//Scorer 7 - Axis positioning relative parameters
scorer7_AxisConfiguration.posRelative.distance := hmiCommands.slitter1.scorerPosCorrectionArr[7].positionCorrection;
scorer7_AxisConfiguration.posRelative.direction := 0;
scorer7_AxisConfiguration.posRelative.velocity := machineConfig.toolSlowPositioningVelocity;
scorer7_AxisConfiguration.posRelative.acceleration := machineConfig.toolSlowPositioningAccel;
scorer7_AxisConfiguration.posRelative.deceleration := machineConfig.toolFastPositioningAccel;
scorer7_AxisConfiguration.posRelative.jerk := machineConfig.toolSlowPositioningJerk;

//Scorer 7 - Axis JOG parameters
scorer7_AxisConfiguration.jog.velocity := machineConfig.toolSlowPositioningVelocity;
scorer7_AxisConfiguration.jog.acceleration := machineConfig.toolSlowPositioningAccel;
scorer7_AxisConfiguration.jog.deceleration := machineConfig.toolFastPositioningAccel;
scorer7_AxisConfiguration.jog.jerk := machineConfig.toolSlowPositioningJerk;

//Scorer 8
//_________________________________________________________________________________________________________________________

scorer8_AxisConfiguration.homing.position := machineConfig.homePositionScorer[8];
scorer8_AxisConfiguration.homing.offsetPosition := machineConfig.homePositionScorer[8];
scorer8_AxisConfiguration.homing.homeExecutionTimeLimit := T#5M;

scorer8_AxisConfiguration.posAbsolute.position := currentOrder.generatedOrder.scorerPositionReferenceArr[8] + machineConfig.scorerPositionCorrectionArr[8];
scorer8_AxisConfiguration.posAbsolute.velocity := machineConfig.toolFastPositioningVelocity;
scorer8_AxisConfiguration.posAbsolute.acceleration := machineConfig.toolFastPositioningAccel;
scorer8_AxisConfiguration.posAbsolute.deceleration := machineConfig.toolFastPositioningDecel;
scorer8_AxisConfiguration.posAbsolute.jerk := machineConfig.toolFastPositioningJerk;

//Scorer 8 - Axis positioning relative parameters
scorer8_AxisConfiguration.posRelative.distance := hmiCommands.slitter1.scorerPosCorrectionArr[8].positionCorrection;
scorer8_AxisConfiguration.posRelative.direction := 0;
scorer8_AxisConfiguration.posRelative.velocity := machineConfig.toolSlowPositioningVelocity;
scorer8_AxisConfiguration.posRelative.acceleration := machineConfig.toolSlowPositioningAccel;
scorer8_AxisConfiguration.posRelative.deceleration := machineConfig.toolFastPositioningAccel;
scorer8_AxisConfiguration.posRelative.jerk := machineConfig.toolSlowPositioningJerk;

//Scorer 8 - Axis JOG parameters
scorer8_AxisConfiguration.jog.velocity := machineConfig.toolSlowPositioningVelocity;
scorer8_AxisConfiguration.jog.acceleration := machineConfig.toolSlowPositioningAccel;
scorer8_AxisConfiguration.jog.deceleration := machineConfig.toolFastPositioningAccel;
scorer8_AxisConfiguration.jog.jerk := machineConfig.toolSlowPositioningJerk;

//----------------------------------------------------------------------------------------------
// Knife Axis control function block calls
//----------------------------------------------------------------------------------------------



IF executePositioning AND NOT executePositioningOld AND homeFinished THEN
//IF executePositioning AND NOT executePositioningOld THEN

	instFbCurrentOrderPositionsGeneration(execute := TRUE,
		machineConfig := machineConfig,
		currentOrder := currentOrder);
			
	IF NOT currentOrder.generatedOrder.statusWord.orderNotOk THEN
		
		instTONExecutePositioningDelay.IN := TRUE;
		positioningStarted	:= TRUE;

	END_IF

END_IF

executePositioningOld := executePositioning;

instTONExecutePositioningDelay(PT:=T#1S);



//Knife 1 - Axis control function block call
//__________________________________________________________________________
instFB_AxisControlKnife1_Axis(
    enable := TRUE,
	fastStop := haltAxis,
    enableAxis := enableAxis,
    resetAxis := resetCmd,
	posAbsolute := instTONExecutePositioningDelay.Q,
	posRelative	:= hmiCommands.slitter1.knifePosCorrectionArr[1].execute,
	jogForward := hmiCommands.slitter1.knifeJogArr[1].jogFw AND NOT homeSensorKnife2 AND homeFinished,
	jogBackward	:= hmiCommands.slitter1.knifeJogArr[1].jogRev AND NOT homeSensorKnife1 AND homeFinished,
    homingSensor := homeSensorKnife1,
    axis := knife1_Axis,
    master := knife1_Axis,
    configuration := knife1_AxisConfiguration
);

//Knife 2 - Axis control function block call
//__________________________________________________________________________

instFB_AxisControlKnife2_Axis(
    enable := TRUE,
	fastStop := haltAxis,	
    enableAxis := enableAxis,
    resetAxis := resetCmd,
	posAbsolute := instTONExecutePositioningDelay.Q,
	posRelative	:= hmiCommands.slitter1.knifePosCorrectionArr[2].execute,
	jogForward := hmiCommands.slitter1.knifeJogArr[2].jogFw AND NOT homeSensorKnife3 AND homeFinished,
	jogBackward	:= hmiCommands.slitter1.knifeJogArr[2].jogRev AND NOT homeSensorKnife2 AND homeFinished,
    homingSensor := homeSensorKnife2,
    axis := knife2_Axis,
    master := knife2_Axis,
    configuration := knife2_AxisConfiguration
);

//Knife 3 - Axis control function block call
//__________________________________________________________________________

instFB_AxisControlKnife3_Axis(
    enable := TRUE,
	fastStop := haltAxis,		
    enableAxis := enableAxis,
    resetAxis := resetCmd,
	posAbsolute := instTONExecutePositioningDelay.Q,
	posRelative	:= hmiCommands.slitter1.knifePosCorrectionArr[3].execute,
	jogForward := hmiCommands.slitter1.knifeJogArr[3].jogFw AND NOT (knife3_Axis.NcToPlc.ActPos > machineConfig.knifeMaxPostionArr[3]) AND NOT limitSensorKnife3_4 AND homeFinished,
	jogBackward	:= hmiCommands.slitter1.knifeJogArr[3].jogRev AND NOT homeSensorKnife3 AND homeFinished,
    homingSensor := homeSensorKnife3,
    axis := knife3_Axis,
    master := knife3_Axis,
    configuration := knife3_AxisConfiguration
);

//Knife 4 - Axis control function block call
//__________________________________________________________________________

instFB_AxisControlKnife4_Axis(
    enable := TRUE,
	fastStop := haltAxis,		
    enableAxis := enableAxis,
    resetAxis := resetCmd,
	posAbsolute := instTONExecutePositioningDelay.Q,
	posRelative	:= hmiCommands.slitter1.knifePosCorrectionArr[4].execute,
	jogForward := hmiCommands.slitter1.knifeJogArr[4].jogFw AND NOT homeSensorKnife4 AND homeFinished,
	jogBackward	:= hmiCommands.slitter1.knifeJogArr[4].jogRev AND NOT (knife4_Axis.NcToPlc.ActPos < machineConfig.knifeMinPostionArr[4]) AND NOT limitSensorKnife3_4 AND homeFinished,
    homingSensor := homeSensorKnife4,
    axis := knife4_Axis,
    master := knife4_Axis,
    configuration := knife4_AxisConfiguration
);

//Knife 5 - Axis control function block call
//__________________________________________________________________________

instFB_AxisControlKnife5_Axis(
    enable := TRUE,
	fastStop := haltAxis,		
    enableAxis := enableAxis,
    resetAxis := resetCmd,
	posAbsolute := instTONExecutePositioningDelay.Q,
	posRelative	:= hmiCommands.slitter1.knifePosCorrectionArr[5].execute,
	jogForward := hmiCommands.slitter1.knifeJogArr[5].jogFw AND NOT homeSensorKnife5 AND homeFinished,
	jogBackward	:= hmiCommands.slitter1.knifeJogArr[5].jogRev AND NOT homeSensorKnife4 AND homeFinished,
    homingSensor := homeSensorKnife5,
    axis := knife5_Axis,
    master := knife5_Axis,
    configuration := knife5_AxisConfiguration
);

//----------------------------------------------------------------------------------------------
// Scorer Axis control function block calls
//----------------------------------------------------------------------------------------------

//Scorer 1
//__________________________________________________________________________

instFB_AxisControlScorer1_Axis(
    enable := TRUE,
	fastStop := haltAxis,		
    enableAxis := enableAxis,
    resetAxis := resetCmd,
	posAbsolute := instTONExecutePositioningDelay.Q,
	posRelative	:= hmiCommands.slitter1.scorerPosCorrectionArr[1].execute,
	jogForward := hmiCommands.slitter1.scorerJogArr[1].jogFw AND NOT homeSensorScorer3 AND homeFinished,
	jogBackward	:= hmiCommands.slitter1.scorerJogArr[1].jogRev AND NOT homeSensorScorer1 AND homeFinished,
    homingSensor := homeSensorScorer1,
    axis := scorer1_Axis,
    master := scorer1_Axis,
    configuration := scorer1_AxisConfiguration
);
//Scorer 2
//__________________________________________________________________________

instFB_AxisControlScorer2_Axis(
    enable := TRUE,
	fastStop := haltAxis,		
    enableAxis := enableAxis,
    resetAxis := resetCmd,
	posAbsolute := instTONExecutePositioningDelay.Q,
	posRelative	:= hmiCommands.slitter1.scorerPosCorrectionArr[2].execute,
	jogForward := hmiCommands.slitter1.scorerJogArr[2].jogFw AND NOT homeSensorScorer4 AND homeFinished,
	jogBackward	:= hmiCommands.slitter1.scorerJogArr[2].jogRev AND NOT homeSensorScorer2 AND homeFinished,
    homingSensor := homeSensorScorer2,
    axis := scorer2_Axis,
    master := scorer2_Axis,
    configuration := scorer2_AxisConfiguration
);

//Scorer 3
//__________________________________________________________________________

instFB_AxisControlScorer3_Axis(
    enable := TRUE,
	fastStop := haltAxis,	
	
    enableAxis := enableAxis,
    resetAxis := resetCmd,
	posAbsolute := instTONExecutePositioningDelay.Q,
	posRelative	:= hmiCommands.slitter1.scorerPosCorrectionArr[3].execute,
	jogForward := hmiCommands.slitter1.scorerJogArr[3].jogFw AND NOT (scorer3_Axis.NcToPlc.ActPos > machineConfig.scorerMaxPostionArr[3]) AND NOT limitSensorScorer3_5 AND homeFinished,
	jogBackward	:= hmiCommands.slitter1.scorerJogArr[3].jogRev AND NOT homeSensorScorer3 AND homeFinished,
    homingSensor := homeSensorScorer3,
    axis := scorer3_Axis,
    master := scorer3_Axis,
    configuration := scorer3_AxisConfiguration
);

//Scorer 4
//__________________________________________________________________________

instFB_AxisControlScorer4_Axis(
    enable := TRUE,
	fastStop := haltAxis,	
	
    enableAxis := enableAxis,
    resetAxis := resetCmd,
	posAbsolute := instTONExecutePositioningDelay.Q,
	posRelative	:= hmiCommands.slitter1.scorerPosCorrectionArr[4].execute,
	jogForward := hmiCommands.slitter1.scorerJogArr[4].jogFw AND NOT (scorer4_Axis.NcToPlc.ActPos > machineConfig.scorerMaxPostionArr[4]) AND NOT limitSensorScorer4_6 AND homeFinished,
	jogBackward	:= hmiCommands.slitter1.scorerJogArr[4].jogRev AND NOT homeSensorScorer4 AND homeFinished,
    homingSensor := homeSensorScorer4,
    axis := scorer4_Axis,
    master := scorer4_Axis,
    configuration := scorer4_AxisConfiguration
);

//Scorer 5
//__________________________________________________________________________

instFB_AxisControlScorer5_Axis(
    enable := TRUE,
	fastStop := haltAxis,	
	
    enableAxis := enableAxis,
    resetAxis := resetCmd,
	posAbsolute := instTONExecutePositioningDelay.Q,
	posRelative	:= hmiCommands.slitter1.scorerPosCorrectionArr[5].execute,
	jogForward := hmiCommands.slitter1.scorerJogArr[5].jogFw AND NOT homeSensorScorer5 AND homeFinished,
	jogBackward	:= hmiCommands.slitter1.scorerJogArr[5].jogRev AND NOT (scorer5_Axis.NcToPlc.ActPos < machineConfig.scorerMinPostionArr[5]) AND NOT limitSensorScorer3_5 AND homeFinished,
    homingSensor := homeSensorScorer5,
    axis := scorer5_Axis,
    master := scorer5_Axis,
    configuration := scorer5_AxisConfiguration
);

//Scorer 6
//__________________________________________________________________________

instFB_AxisControlScorer6_Axis(
    enable := TRUE,
	fastStop := haltAxis,	
	
    enableAxis := enableAxis,
    resetAxis := resetCmd,
	posAbsolute := instTONExecutePositioningDelay.Q,
	posRelative	:= hmiCommands.slitter1.scorerPosCorrectionArr[6].execute,
	jogForward := hmiCommands.slitter1.scorerJogArr[6].jogFw AND NOT homeSensorScorer6 AND homeFinished,
	jogBackward	:= hmiCommands.slitter1.scorerJogArr[6].jogRev AND NOT (scorer6_Axis.NcToPlc.ActPos < machineConfig.scorerMinPostionArr[6]) AND NOT limitSensorScorer4_6 AND homeFinished,
    homingSensor := homeSensorScorer6,
    axis := scorer6_Axis,
    master := scorer6_Axis,
    configuration := scorer6_AxisConfiguration
);

//Scorer 7
//__________________________________________________________________________

instFB_AxisControlScorer7_Axis(
    enable := TRUE,
	fastStop := haltAxis,	
	
    enableAxis := enableAxis,
    resetAxis := resetCmd,
	posAbsolute := instTONExecutePositioningDelay.Q,
	posRelative	:= hmiCommands.slitter1.scorerPosCorrectionArr[7].execute,
	jogForward := hmiCommands.slitter1.scorerJogArr[7].jogFw AND NOT homeSensorScorer7 AND homeFinished,
	jogBackward	:= hmiCommands.slitter1.scorerJogArr[7].jogRev AND NOT homeSensorScorer5 AND homeFinished,
    homingSensor := homeSensorScorer7,
    axis := scorer7_Axis,
    master := scorer7_Axis,
    configuration := scorer7_AxisConfiguration
);

//Scorer 8
//__________________________________________________________________________

instFB_AxisControlScorer8_Axis(
    enable := TRUE,
	fastStop := haltAxis,	
	
    enableAxis := enableAxis,
    resetAxis := resetCmd,
	posAbsolute := instTONExecutePositioningDelay.Q,
	posRelative	:= hmiCommands.slitter1.scorerPosCorrectionArr[8].execute,
	jogForward := hmiCommands.slitter1.scorerJogArr[8].jogFw AND NOT homeSensorScorer8 AND homeFinished,
	jogBackward	:= hmiCommands.slitter1.scorerJogArr[8].jogRev AND NOT homeSensorScorer6 AND homeFinished,
    homingSensor := homeSensorScorer8,
    axis := scorer8_Axis,
    master := scorer8_Axis,
    configuration := scorer8_AxisConfiguration
);

IF instTONExecutePositioningDelay.Q THEN
	
	instTONExecutePositioningDelay.IN := FALSE;
	positioningStarted	:= FALSE;


END_IF
END_METHOD

METHOD PRIVATE _exhaustMotor
VAR_INPUT
END_VAR
(*
	startExhaustMotorCmd				: BOOL;
	stopExhaustMotorCmd				: BOOL;

*)

IF startExhaustMotorCmd AND safetyOK THEN
	
	startExhaustMotor := TRUE;


END_IF

IF stopExhaustMotorCmd THEN
	
	startExhaustMotor := FALSE;

END_IF



startExhaustMotorLamp := startExhaustMotor;
END_METHOD

METHOD PRIVATE _haltTheAxis
VAR_INPUT
END_VAR
(*

	homeSensorKnife1					: BOOL; // Knife 1 - Home sensor
	homeSensorKnife2					: BOOL; // Knife 2 - Home sensor
	homeSensorKnife3					: BOOL; // Knife 3 - Home sensor
	homeSensorKnife4					: BOOL; // Knife 4 - Home sensor
	homeSensorKnife5					: BOOL; // Knife 5 - Home sensor
	
	homeSensorScorer1					: BOOL; // Scorer 1 - Home sensor
	homeSensorScorer2					: BOOL; // Scorer 1 - Home sensor
	homeSensorScorer3					: BOOL; // Scorer 1 - Home sensor
	homeSensorScorer4					: BOOL; // Scorer 1 - Home sensor
	homeSensorScorer5					: BOOL; // Scorer 1 - Home sensor
	homeSensorScorer6					: BOOL; // Scorer 1 - Home sensor
	homeSensorScorer7					: BOOL; // Scorer 1 - Home sensor
	homeSensorScorer8					: BOOL; // Scorer 1 - Home sensor
*)

(*

	limitSensorKnife3_4					: BOOL;
	limitSensorScorer4_6					: BOOL;
	limitSensorScorer3_5					: BOOL;
*)
//-------------------------------------------------------------------------------------------------
// Halt Axis Logic: Prevent motion if any tool is detected on home sensor during active positioning
//-------------------------------------------------------------------------------------------------

// Activate the halt trigger if positioning is in progress 
// and any knife or scorer is detected in the home sensor
IF positioningRunning AND (
     homeSensorKnife1 OR
     homeSensorKnife2 OR
     homeSensorKnife3 OR
     homeSensorKnife4 OR
     homeSensorKnife5 OR
     homeSensorScorer1 OR
     homeSensorScorer2 OR
     homeSensorScorer3 OR
     homeSensorScorer4 OR
     homeSensorScorer5 OR
     homeSensorScorer6 OR
     homeSensorScorer7 OR
     homeSensorScorer8 OR
	 limitSensorKnife3_4 OR
	 limitSensorScorer3_5 OR
 	 limitSensorScorer4_6 
	 
) THEN
    instTPHaltAxis.IN := TRUE;
ELSE
    instTPHaltAxis.IN := FALSE;
END_IF

// Timer pulse for halting signal - triggers TRUE for 1 second
instTPHaltAxis(PT := T#1S);

// Output signal to halt all axes
haltAxis := instTPHaltAxis.Q;
END_METHOD

METHOD _homeFinished
VAR_INPUT
END_VAR
homeFinished := knife1_Axis.Status.Homed AND knife2_Axis.Status.Homed AND knife3_Axis.Status.Homed AND knife4_Axis.Status.Homed AND knife5_Axis.Status.Homed AND scorer1_Axis.Status.Homed AND scorer2_Axis.Status.Homed AND scorer3_Axis.Status.Homed AND scorer4_Axis.Status.Homed AND scorer5_Axis.Status.Homed AND scorer6_Axis.Status.Homed AND scorer7_Axis.Status.Homed AND scorer8_Axis.Status.Homed;
END_METHOD

METHOD PRIVATE _knifeLubrification
VAR_INPUT
END_VAR


(*
	knifeRunningMetersForSharpening		: ARRAY [1..5] OF INT;	(*This array is used to reset the lifetime meters that the knife runs*)
	knifeRunningMetersForLubfrication		: ARRAY [1..5] OF INT;	(*This array is used to reset the lifetime meters that the knife runs*)
	

*)

knifeLubrificationPump := startCutting;


instKnifeLubrificationCLK_PRG(PT:= T#1S, Q=> );


inst_FB_KnifeLubrification[1](
	machineRunning:= startTractionMotorCmd AND startCutting,
	manualLubrification := knife1LubrificationCmd, 
	measuringWheelSensor:= measuringWheelPulseSensor, 
	knifeEnabled:= knife1Enabled, 
	lubrificationSetpoint := machineConfig.knifeLubrificationDistance, 
	lubrificationTime:= machineConfig.knifeLubrificationTime, 
	lubrificationSolenoid=> knife1Lubrification);
	
inst_FB_KnifeLubrification[2](
	machineRunning:= startTractionMotorCmd AND startCutting,
	manualLubrification := knife2LubrificationCmd,  
	measuringWheelSensor:= measuringWheelPulseSensor, 
	knifeEnabled:= knife2Enabled, 
	lubrificationSetpoint := machineConfig.knifeLubrificationDistance, 
	lubrificationTime:= machineConfig.knifeLubrificationTime, 
	lubrificationSolenoid=> knife2Lubrification);
	
inst_FB_KnifeLubrification[3](
	machineRunning:= startTractionMotorCmd AND startCutting, 
	manualLubrification := knife3LubrificationCmd, 
	measuringWheelSensor:= measuringWheelPulseSensor, 
	knifeEnabled:= knife3Enabled, 
	lubrificationSetpoint := machineConfig.knifeLubrificationDistance, 
	lubrificationTime:= machineConfig.knifeLubrificationTime, 
	lubrificationSolenoid=> knife3Lubrification);	
	
inst_FB_KnifeLubrification[4](
	machineRunning:= startTractionMotorCmd AND startCutting, 
	manualLubrification := knife4LubrificationCmd, 	
	measuringWheelSensor:= measuringWheelPulseSensor, 
	knifeEnabled:= knife4Enabled, 
	lubrificationSetpoint := machineConfig.knifeLubrificationDistance, 
	lubrificationTime:= machineConfig.knifeLubrificationTime, 
	lubrificationSolenoid=> knife4Lubrification);		
	
	
inst_FB_KnifeLubrification[5](
	machineRunning:= startTractionMotorCmd AND startCutting, 
	manualLubrification := knife5LubrificationCmd,  
	measuringWheelSensor:= measuringWheelPulseSensor, 
	knifeEnabled:= knife5Enabled,
	lubrificationSetpoint := machineConfig.knifeLubrificationDistance, 
	lubrificationTime:= machineConfig.knifeLubrificationTime, 
	lubrificationSolenoid=> knife5Lubrification);		
	
arrKnifeRunningMetersForLubfrication[1] := inst_FB_KnifeLubrification[1].knifeRunningMeters;	
arrKnifeRunningMetersForLubfrication[2] := inst_FB_KnifeLubrification[2].knifeRunningMeters;	
arrKnifeRunningMetersForLubfrication[3] := inst_FB_KnifeLubrification[3].knifeRunningMeters;	
arrKnifeRunningMetersForLubfrication[4] := inst_FB_KnifeLubrification[4].knifeRunningMeters;	
arrKnifeRunningMetersForLubfrication[5] := inst_FB_KnifeLubrification[5].knifeRunningMeters;
END_METHOD

METHOD PRIVATE _knifeSharpening
VAR_INPUT
END_VAR
(*
	knifeRunningMetersForSharpening		: ARRAY [1..5] OF INT;	(*This array is used to reset the lifetime meters that the knife runs*)
	knifeRunningMetersForLubfrication		: ARRAY [1..5] OF INT;	(*This array is used to reset the lifetime meters that the knife runs*)
	

*)
//=================================================================================================
// KNIFE SHARPENING FB CALLS (1..7)
//=================================================================================================

inst_FB_KnifeSharpening[1](
    machineRunning        := knifeMotorStart,
    manualSharpening      := knifeManualSharpeningCmdArr[1],
    measuringWheelSensor  := measuringWheelPulseSensor,
    knifeEnabled          := currentOrder.generatedOrder.knifeEnabledArr[1],
    sharpeningSetpoint    := machineConfig.knifeSharpeningDistance,
    sharpeningTime        := machineConfig.knifeSharpeningTimeMS,
    sharpeningSolenoid    => knife1Sharpening
);

inst_FB_KnifeSharpening[2](
    machineRunning        := knifeMotorStart,
    manualSharpening      := knifeManualSharpeningCmdArr[2],
    measuringWheelSensor  := measuringWheelPulseSensor,
    knifeEnabled          := currentOrder.generatedOrder.knifeEnabledArr[2],
    sharpeningSetpoint    := machineConfig.knifeSharpeningDistance,
    sharpeningTime        := machineConfig.knifeSharpeningTimeMS,
    sharpeningSolenoid    => knife2Sharpening
);

inst_FB_KnifeSharpening[3](
    machineRunning        := knifeMotorStart,
    manualSharpening      := knifeManualSharpeningCmdArr[3],
    measuringWheelSensor  := measuringWheelPulseSensor,
    knifeEnabled          := currentOrder.generatedOrder.knifeEnabledArr[3],
    sharpeningSetpoint    := machineConfig.knifeSharpeningDistance,
    sharpeningTime        := machineConfig.knifeSharpeningTimeMS,
    sharpeningSolenoid    => knife3Sharpening
);

inst_FB_KnifeSharpening[4](
    machineRunning        := knifeMotorStart,
    manualSharpening      := knifeManualSharpeningCmdArr[4],
    measuringWheelSensor  := measuringWheelPulseSensor,
    knifeEnabled          := currentOrder.generatedOrder.knifeEnabledArr[4],
    sharpeningSetpoint    := machineConfig.knifeSharpeningDistance,
    sharpeningTime        := machineConfig.knifeSharpeningTimeMS,
    sharpeningSolenoid    => knife4Sharpening
);

inst_FB_KnifeSharpening[5](
    machineRunning        := knifeMotorStart,
    manualSharpening      := knifeManualSharpeningCmdArr[5],
    measuringWheelSensor  := measuringWheelPulseSensor,
    knifeEnabled          := currentOrder.generatedOrder.knifeEnabledArr[5],
    sharpeningSetpoint    := machineConfig.knifeSharpeningDistance,
    sharpeningTime        := machineConfig.knifeSharpeningTimeMS,
    sharpeningSolenoid    => knife5Sharpening
);
END_METHOD

METHOD PRIVATE _knifeSharpening_old
VAR_INPUT
END_VAR
(*
	knifeRunningMetersForSharpening		: ARRAY [1..5] OF INT;	(*This array is used to reset the lifetime meters that the knife runs*)
	knifeRunningMetersForLubfrication		: ARRAY [1..5] OF INT;	(*This array is used to reset the lifetime meters that the knife runs*)
	
	paperPresenceSensor				: BOOL;
	measuringWheelPaperPresenceSensor		: BOOL;
	rotaryShearCutPulse					: BOOL;	
	measuringWheelPulseSensor		: BOOL;	

*)

IF NOT knifeSharpeningAutoMan THEN
	
	knife1Sharpening := knife1SharpeningCmd;
	knife2Sharpening := knife2SharpeningCmd;
	knife3Sharpening := knife3SharpeningCmd;
	knife4Sharpening := knife4SharpeningCmd;
	knife5Sharpening := knife5SharpeningCmd;
	
	knife1SharpeningLamp := knife1Sharpening;
	knife2SharpeningLamp := knife2Sharpening;
	knife3SharpeningLamp := knife3Sharpening;
	knife4SharpeningLamp := knife4Sharpening;
	knife5SharpeningLamp := knife5Sharpening;	

ELSE	
;


instKnifeSharpeningCLK_PRG(PT:= T#1S, Q=> );


inst_FB_KnifeSharpening[1](
	machineRunning:= startTractionMotorCmd AND startCutting, 
	manualSharpening:= knife1SharpeningCmd, 
	measuringWheelSensor:= measuringWheelPulseSensor, 
	knifeEnabled:= knife1Enabled, 
	sharpeningSetpoint:= machineConfig.knifeSharpeningDistance, 
	sharpeningTime:= machineConfig.knifeSharpeningTime, 
	sharpeningSolenoid=> knife1Sharpening);


inst_FB_KnifeSharpening[2](
	machineRunning:= startTractionMotorCmd AND startCutting, 
	manualSharpening:= knife2SharpeningCmd, 
	measuringWheelSensor:= measuringWheelPulseSensor, 
	knifeEnabled:= knife2Enabled, 
	sharpeningSetpoint:= machineConfig.knifeSharpeningDistance, 
	sharpeningTime:= machineConfig.knifeSharpeningTime, 
	sharpeningSolenoid=> knife2Sharpening);	
	
inst_FB_KnifeSharpening[3](
	machineRunning:= startTractionMotorCmd AND startCutting, 
	manualSharpening:= knife3SharpeningCmd, 
	measuringWheelSensor:= measuringWheelPulseSensor, 
	knifeEnabled:= knife3Enabled, 
	sharpeningSetpoint:= machineConfig.knifeSharpeningDistance, 
	sharpeningTime:= machineConfig.knifeSharpeningTime, 
	sharpeningSolenoid=> knife3Sharpening);	

inst_FB_KnifeSharpening[4](
	machineRunning:= startTractionMotorCmd AND startCutting, 
	manualSharpening:= knife4SharpeningCmd, 
	measuringWheelSensor:= measuringWheelPulseSensor, 
	knifeEnabled:= knife4Enabled, 
	sharpeningSetpoint:= machineConfig.knifeSharpeningDistance, 
	sharpeningTime:= machineConfig.knifeSharpeningTime, 
	sharpeningSolenoid=> knife4Sharpening);	


inst_FB_KnifeSharpening[5](
	machineRunning:= startTractionMotorCmd AND startCutting, 
	manualSharpening:= knife5SharpeningCmd, 
	measuringWheelSensor:= measuringWheelPulseSensor, 
	knifeEnabled:= knife5Enabled, 
	sharpeningSetpoint:= machineConfig.knifeSharpeningDistance, 
	sharpeningTime:= machineConfig.knifeSharpeningTime, 
	sharpeningSolenoid=> knife5Sharpening);		

END_IF


arrKnifeRunningMetersForSharpening[1] := inst_FB_KnifeSharpening[1].knifeRunningMeters;
arrKnifeRunningMetersForSharpening[2] := inst_FB_KnifeSharpening[2].knifeRunningMeters;
arrKnifeRunningMetersForSharpening[3] := inst_FB_KnifeSharpening[3].knifeRunningMeters;
arrKnifeRunningMetersForSharpening[4] := inst_FB_KnifeSharpening[4].knifeRunningMeters;
arrKnifeRunningMetersForSharpening[5] := inst_FB_KnifeSharpening[5].knifeRunningMeters;
END_METHOD

METHOD PRIVATE _paperDirectionFlaps
VAR_INPUT
END_VAR
(*

	paperDirectionFlapAutoMan	: BOOL; // Paper direction flap (0=Manual / 1=Auto)
    paperDirectionFlap01Cmd    : BOOL;
	
	rotaryKnifeInfeedUpperDamper1Cmd : BOOL;
	rotaryKnifeInfeedUpperDamper2Cmd : BOOL;
	
	rotaryKnifeInfeedLowerDamper1Cmd : BOOL;
	rotaryKnifeInfeedLowerDamper2Cmd : BOOL;
	
	pilotRollUpDownCmd			: BOOL;
	
	
*)

IF NOT paperDirectionFlapAutoMan THEN
	
	paperDirectionFlap01 := paperDirectionFlap01Cmd;
	paperDirectionFlap02 := paperDirectionFlap02Cmd;
	paperDirectionFlap03 := paperDirectionFlap03Cmd;
	paperDirectionFlap04 := paperDirectionFlap04Cmd;
	paperDirectionFlap05 := paperDirectionFlap05Cmd;
	paperDirectionFlap06 := paperDirectionFlap06Cmd;
	paperDirectionFlap07 := paperDirectionFlap07Cmd;
	paperDirectionFlap08 := paperDirectionFlap08Cmd;
	paperDirectionFlap09 := paperDirectionFlap09Cmd;
	paperDirectionFlap10 := paperDirectionFlap10Cmd;
	paperDirectionFlap11 := paperDirectionFlap11Cmd;
	paperDirectionFlap12 := paperDirectionFlap12Cmd;
	
ELSE
	;
END_IF



rotaryKnifeInfeedUpperDamper1 := rotaryKnifeInfeedUpperDamper1Cmd;
rotaryKnifeInfeedUpperDamper2 := rotaryKnifeInfeedUpperDamper2Cmd;

rotaryKnifeInfeedLowerDamper1 := rotaryKnifeInfeedLowerDamper1Cmd;
rotaryKnifeInfeedLowerDamper2 := rotaryKnifeInfeedLowerDamper2Cmd;

pilotRollUpDown := pilotRollUpDownCmd;
END_METHOD

METHOD PRIVATE _paperTrim
VAR_INPUT
END_VAR



	    // Paper scrap controls
    paperTrimOperatorSideOpen  := paperTrimOperatorSideOpenCmd AND NOT paperTrimOperatorSideCloseCmd AND safetyOK;
    paperTrimOperatorSideClose := paperTrimOperatorSideCloseCmd AND NOT paperTrimOperatorSideOpenCmd AND safetyOK;
    paperTrimMotorSideOpen     := paperTrimMotorSideOpenCmd AND NOT paperTrimMotorSideCloseCmd AND safetyOK;
    paperTrimMotorSideClose    := paperTrimMotorSideCloseCmd AND NOT paperTrimMotorSideOpenCmd AND safetyOK;
END_METHOD

METHOD _safetyCircuit : BOOL
VAR_INPUT
END_VAR
safetyOK := safetyFeedback;


safetyOKLamp := NOT safetyOK;
END_METHOD

METHOD PRIVATE _scorerHeightControl

VAR CONSTANT

    STATE_MANUAL : INT := 0;

    STATE_GOTO_D : INT := 1;
    STATE_WAIT_D : INT := 2;

    STATE_GOTO_W : INT := 3;
    STATE_WAIT_W : INT := 4;

    STATE_GOTO_N : INT := 5;
    STATE_WAIT_N : INT := 6;
END_VAR

{===== Rising-edge commands =====}
IF scorerTypeDCmd AND NOT scorerTypeDCmdOld THEN
    scorerHeightPositioningState := STATE_GOTO_D;
END_IF;
scorerTypeDCmdOld := scorerTypeDCmd;

IF scorerTypeWCmd AND NOT scorerTypeWCmdOld THEN
    scorerHeightPositioningState := STATE_GOTO_W;
END_IF;
scorerTypeWCmdOld := scorerTypeWCmd;   // <-- fixed (was assigning N old flag before)

IF scorerTypeNCmd AND NOT scorerTypeNCmdOld THEN
    scorerHeightPositioningState := STATE_GOTO_N;
END_IF;
scorerTypeNCmdOld := scorerTypeNCmd;


IF NOT safetyOK THEN
	
	scorerHeightPositioningState := 0;

END_IF


{===== State machine =====}
CASE scorerHeightPositioningState OF

    // -------------------------------------------------------------
    // 0) MANUAL CONTROL
    //    Pass-through of manual jog commands to the motor.
    // -------------------------------------------------------------
    STATE_MANUAL:
        scorerHeightPositioningRunning := FALSE;

        // Manual jog direction
        scorerHeightInc := scorerHeightIncCmd;
        scorerHeightDec := scorerHeightDecCmd;

        // Manual speed (both TRUE here = slow; adjust if you have a separate speed scheme)
        scorerHeightMotorStart := (scorerHeightInc OR scorerHeightDec) AND safetyOK;
        scorerHeightMotorSlow  := (scorerHeightInc OR scorerHeightDec) AND safetyOK;
        scorerHeightMotorFast  := FALSE;



    // -------------------------------------------------------------
    // 1) SELECT D — START MOVE (fast up)
    // -------------------------------------------------------------
    STATE_GOTO_D:
        scorerHeightPositioningRunning := TRUE;

        // Lamps while moving: blink only the requested type
        scorerTypeDLamp := FALSE;   // will blink in WAIT state
        scorerTypeWLamp := FALSE;
        scorerTypeNLamp := FALSE;

        // Start motion
        scorerHeightMotorStart := TRUE;
        scorerHeightMotorFast  := TRUE;
        scorerHeightMotorSlow  := FALSE;

        // Direction to reach the D height (set per your mechanics)
        scorerHeightInc := TRUE;
        scorerHeightDec := FALSE;

        // Start settle timer (TOF)
        instTOFScorerSensorDelay(IN := TRUE);

        // Next
        scorerHeightPositioningState := STATE_WAIT_D;


    // -------------------------------------------------------------
    // 2) SELECT D — WAIT FOR SENSOR AFTER DELAY
    // -------------------------------------------------------------
    STATE_WAIT_D:
        instTOFScorerSensorDelay.IN := FALSE;     // start counting off-delay
        scorerTypeDLamp := clock_Pulse_1S;        // blink while seeking

        // Accept sensor only after the off-delay has elapsed (Q = FALSE)
        IF scorerTypeDSensor AND NOT instTOFScorerSensorDelay.Q THEN
            // Stop motion
            scorerHeightMotorStart := FALSE;
            scorerHeightMotorFast  := FALSE;
            scorerHeightMotorSlow  := FALSE;

            scorerHeightInc := FALSE;
            scorerHeightDec := FALSE;

            // Solid lamp for selected type
            scorerTypeDLamp := TRUE;
            scorerTypeWLamp := FALSE;
            scorerTypeNLamp := FALSE;

            // Return to manual
            scorerHeightPositioningState := STATE_MANUAL;
        END_IF;


    // -------------------------------------------------------------
    // 3) SELECT W — START MOVE (fast up)
    // -------------------------------------------------------------
    STATE_GOTO_W:
        scorerHeightPositioningRunning := TRUE;

        scorerTypeDLamp := FALSE;
        scorerTypeWLamp := FALSE;   // will blink in WAIT state
        scorerTypeNLamp := FALSE;

        scorerHeightMotorStart := TRUE;
        scorerHeightMotorFast  := TRUE;
        scorerHeightMotorSlow  := FALSE;

        scorerHeightInc := TRUE;    // adjust direction if your mechanics require
        scorerHeightDec := FALSE;

        instTOFScorerSensorDelay(IN := TRUE);

        scorerHeightPositioningState := STATE_WAIT_W;


    // -------------------------------------------------------------
    // 4) SELECT W — WAIT FOR SENSOR AFTER DELAY
    // -------------------------------------------------------------
    STATE_WAIT_W:
        instTOFScorerSensorDelay.IN := FALSE;
        scorerTypeWLamp := clock_Pulse_1S;

        IF scorerTypeWSensor AND NOT instTOFScorerSensorDelay.Q THEN
            scorerHeightMotorStart := FALSE;
            scorerHeightMotorFast  := FALSE;
            scorerHeightMotorSlow  := FALSE;

            scorerHeightInc := FALSE;
            scorerHeightDec := FALSE;

            scorerTypeDLamp := FALSE;
            scorerTypeWLamp := TRUE;
            scorerTypeNLamp := FALSE;

            scorerHeightPositioningState := STATE_MANUAL;
        END_IF;


    // -------------------------------------------------------------
    // 5) SELECT N — START MOVE (fast up)
    // -------------------------------------------------------------
    STATE_GOTO_N:
        scorerHeightPositioningRunning := TRUE;

        scorerTypeDLamp := FALSE;
        scorerTypeWLamp := FALSE;
        scorerTypeNLamp := FALSE;   // will blink in WAIT state

        scorerHeightMotorStart := TRUE;
        scorerHeightMotorFast  := TRUE;
        scorerHeightMotorSlow  := FALSE;

        scorerHeightInc := TRUE;    // adjust if needed
        scorerHeightDec := FALSE;

        instTOFScorerSensorDelay(IN := TRUE);

        scorerHeightPositioningState := STATE_WAIT_N;


    // -------------------------------------------------------------
    // 6) SELECT N — WAIT FOR SENSOR AFTER DELAY
    // -------------------------------------------------------------
    STATE_WAIT_N:
        instTOFScorerSensorDelay.IN := FALSE;
        scorerTypeNLamp := clock_Pulse_1S;

        IF scorerTypeNSensor AND NOT instTOFScorerSensorDelay.Q THEN
            scorerHeightMotorStart := FALSE;
            scorerHeightMotorFast  := FALSE;
            scorerHeightMotorSlow  := FALSE;

            scorerHeightInc := FALSE;
            scorerHeightDec := FALSE;

            scorerTypeDLamp := FALSE;
            scorerTypeWLamp := FALSE;
            scorerTypeNLamp := TRUE;

            scorerHeightPositioningState := STATE_MANUAL;
        END_IF;


    // -------------------------------------------------------------
    // SAFETY FALLBACK
    // -------------------------------------------------------------
    ELSE
        // Any undefined state: stop and drop back to manual
        scorerHeightMotorStart := FALSE;
        scorerHeightMotorFast  := FALSE;
        scorerHeightMotorSlow  := FALSE;

        scorerHeightInc := FALSE;
        scorerHeightDec := FALSE;

        scorerHeightPositioningState := STATE_MANUAL;
END_CASE;


{===== Timers / Blink generator configuration =====}
instTOFScorerSensorDelay(PT := T#3S);  // settle / anti-bounce window
inst_GEN_PULSE_1S(ENQ := TRUE, PTH := T#1S, PTL := T#1S, Q => clock_Pulse_1S);
END_METHOD

METHOD PRIVATE _slitterCenterPaperGuideRoll
VAR_INPUT
END_VAR




slitterCenterGuideRoll := slitterCenterGuideRollCmd;
END_METHOD

METHOD PRIVATE _slitterDisplacement
VAR_INPUT
END_VAR
(*
    moveSlitterOperatorSideLimit : BOOL;
    moveSlitterMotorSideLimit    : BOOL;

*)
    // Slitter movement controls
moveSlitterOperatorSide :=	moveSlitterOperatorSideCmd AND NOT moveSlitterMotorSideCmd AND moveSlitterOperatorSideLimit AND safetyOK;
moveSlitterMotorSide :=	moveSlitterMotorSideCmd   AND NOT moveSlitterOperatorSideCmd AND moveSlitterMotorSideLimit AND safetyOK;

moveSlitterOperatorSideLamp := moveSlitterOperatorSide;
moveSlitterMotorSideLamp    := moveSlitterMotorSide;
END_METHOD

METHOD _slitterPaperDirectionControl
// Call the Function Block (Execute when the positioning finishes)

//Check for rising edge
instRTrigToolsInPosition(CLK := bAllKnivesInPos);


//Confirm the current order position before set the flap positions
IF hmiCommands.slitter1.flapsSetAuto AND NOT flapsSetAutoOld THEN
	
	
	instFbCurrentOrderPositionsGeneration(execute := TRUE,
		machineConfig := machineConfig,
		currentOrder := currentOrder);
	
END_IF
flapsSetAutoOld := hmiCommands.slitter1.flapsSetAuto;

instFB_PaperDirectionControl(
	executeCmd := instRTrigToolsInPosition.Q OR hmiCommands.slitter1.flapsSetAuto,
	allUPCmd := hmiCommands.slitter1.flapsAllUP,
	allDownCmd := hmiCommands.slitter1.flapsAllDown,
	invertDirection := hmiCommands.slitter1.flapsInvertDirection,
    currentOrder  := currentOrder, 
    machineConfig := machineConfig,
	flapsManualCmdArr := flapsManualCmdArr
);


// Map internal array to physical output variables
paperDirectionFlap01 := NOT instFB_PaperDirectionControl.flapSolenoidArr[1];
paperDirectionFlap02 := NOT instFB_PaperDirectionControl.flapSolenoidArr[2];
paperDirectionFlap03 := NOT instFB_PaperDirectionControl.flapSolenoidArr[3];
paperDirectionFlap04 := NOT instFB_PaperDirectionControl.flapSolenoidArr[4];
paperDirectionFlap05 := NOT instFB_PaperDirectionControl.flapSolenoidArr[5];
paperDirectionFlap06 := NOT instFB_PaperDirectionControl.flapSolenoidArr[6];
paperDirectionFlap07 := NOT instFB_PaperDirectionControl.flapSolenoidArr[7];
paperDirectionFlap08 := NOT instFB_PaperDirectionControl.flapSolenoidArr[8];
paperDirectionFlap09 := NOT instFB_PaperDirectionControl.flapSolenoidArr[9];
paperDirectionFlap10 := NOT instFB_PaperDirectionControl.flapSolenoidArr[10];
paperDirectionFlap11 := NOT instFB_PaperDirectionControl.flapSolenoidArr[11];
paperDirectionFlap12 := NOT instFB_PaperDirectionControl.flapSolenoidArr[12];
END_METHOD

METHOD PRIVATE _startStopCutting
VAR_INPUT
END_VAR
IF startCuttingCmd THEN
	
	startCutting := TRUE;

END_IF

IF stopCuttingCmd THEN
	
	startCutting := FALSE;;

END_IF


startCuttingLamp := startCutting;
END_METHOD

METHOD _startTractionMotor
VAR_INPUT
END_VAR
IF startTractionMotorCmd AND safetyOK THEN
	
    // Motor commands
    knifeMotorStart         := TRUE;
    scorerMotorStart        := TRUE;
	tractionEnabledLamp		:= TRUE;
ELSE
	
    // Motor commands
    knifeMotorStart         := FALSE;
    scorerMotorStart        := FALSE;
	tractionEnabledLamp		:= FALSE;	
	
END_IF

	
	IF NOT aocRunning THEN
	
			slitterKnifeDriveRef := LIMIT(machineConfig.minLineSpeed,
										  lineSpeedMPM,
										  999) * machineConfig.knifeSpeedOffset;	
			
			slitterScorerDriveRef := LIMIT(machineConfig.minLineSpeed,
										  lineSpeedMPM,
										  999) * machineConfig.scorerSpeedOffset;		
		
		ELSE
		
			slitterKnifeDriveRef := LIMIT(machineConfig.minLineSpeed,
										  aocSpeedMPM,
										  999) * machineConfig.knifeSpeedOffset;	
			
			slitterScorerDriveRef := LIMIT(machineConfig.minLineSpeed,
										  aocSpeedMPM,
										  999) * machineConfig.scorerSpeedOffset;			
		
		END_IF


    // Zero references when drives are not commanded to run to prevent stale setpoints
IF NOT knifeMotorStart THEN
	slitterKnifeDriveRef := 0.0;
END_IF;

IF NOT scorerMotorStart THEN
	slitterScorerDriveRef := 0.0;
END_IF;
END_METHOD

METHOD PRIVATE _toolEnabledLamp
VAR_INPUT
END_VAR
knife1EnabledLamp :=  knife1Enabled;
knife2EnabledLamp :=  knife2Enabled;
knife3EnabledLamp :=  knife3Enabled;
knife4EnabledLamp :=  knife4Enabled;
knife5EnabledLamp :=  knife5Enabled;

scorer1EnabledLamp := scorer1Enabled;
scorer2EnabledLamp := scorer2Enabled;
scorer3EnabledLamp := scorer3Enabled;
scorer4EnabledLamp := scorer4Enabled;
scorer5EnabledLamp := scorer5Enabled;
scorer6EnabledLamp := scorer6Enabled;
scorer7EnabledLamp := scorer7Enabled;
scorer8EnabledLamp := scorer8Enabled;
END_METHOD

METHOD PRIVATE _toolsUpDownControl
VAR_INPUT
END_VAR
(*
	knife1Enabled						: BOOL;	//Knife 1 - Solenoid enabled
	knife2Enabled						: BOOL;	//Knife 1 - Solenoid enabled
	knife3Enabled						: BOOL;	//Knife 1 - Solenoid enabled
	knife4Enabled						: BOOL;	//Knife 1 - Solenoid enabled
	knife5Enabled						: BOOL;	//Knife 1 - Solenoid enabled

	scorer1Enabled						: BOOL;	//Scorer 1 - Solenoid enabled
	scorer2Enabled						: BOOL;	//Scorer 2 - Solenoid enabled
	scorer3Enabled						: BOOL;	//Scorer 3 - Solenoid enabled
	scorer4Enabled						: BOOL;	//Scorer 4 - Solenoid enabled
	scorer5Enabled						: BOOL;	//Scorer 5 - Solenoid enabled
	scorer6Enabled						: BOOL;	//Scorer 6 - Solenoid enabled
	scorer7Enabled						: BOOL;	//Scorer 7 - Solenoid enabled
	scorer8Enabled						: BOOL;	//Scorer 8 - Solenoid enabled*)
VAR

END_VAR
// ===================== KNIFES 1..5 =====================
IF knife1EnabledCmd AND NOT knife1EnabledCmdOld THEN
    IF currentOrder.generatedOrder.knifeEnabledArr[1] THEN
        currentOrder.generatedOrder.knifeEnabledArr[1] := FALSE;
    ELSE
        currentOrder.generatedOrder.knifeEnabledArr[1] := TRUE;
    END_IF
END_IF
knife1EnabledCmdOld := knife1EnabledCmd;

IF knife2EnabledCmd AND NOT knife2EnabledCmdOld THEN
    IF currentOrder.generatedOrder.knifeEnabledArr[2] THEN
        currentOrder.generatedOrder.knifeEnabledArr[2] := FALSE;
    ELSE
        currentOrder.generatedOrder.knifeEnabledArr[2] := TRUE;
    END_IF
END_IF
knife2EnabledCmdOld := knife2EnabledCmd;

IF knife3EnabledCmd AND NOT knife3EnabledCmdOld THEN
    IF currentOrder.generatedOrder.knifeEnabledArr[3] THEN
        currentOrder.generatedOrder.knifeEnabledArr[3] := FALSE;
    ELSE
        currentOrder.generatedOrder.knifeEnabledArr[3] := TRUE;
    END_IF
END_IF
knife3EnabledCmdOld := knife3EnabledCmd;

IF knife4EnabledCmd AND NOT knife4EnabledCmdOld THEN
    IF currentOrder.generatedOrder.knifeEnabledArr[4] THEN
        currentOrder.generatedOrder.knifeEnabledArr[4] := FALSE;
    ELSE
        currentOrder.generatedOrder.knifeEnabledArr[4] := TRUE;
    END_IF
END_IF
knife4EnabledCmdOld := knife4EnabledCmd;

IF knife5EnabledCmd AND NOT knife5EnabledCmdOld THEN
    IF currentOrder.generatedOrder.knifeEnabledArr[5] THEN
        currentOrder.generatedOrder.knifeEnabledArr[5] := FALSE;
    ELSE
        currentOrder.generatedOrder.knifeEnabledArr[5] := TRUE;
    END_IF
END_IF
knife5EnabledCmdOld := knife5EnabledCmd;


// ===================== SCORERS 1..8 =====================
IF scorer1EnabledCmd AND NOT scorer1EnabledCmdOld THEN
    IF currentOrder.generatedOrder.scorerEnabledArr[1] THEN
        currentOrder.generatedOrder.scorerEnabledArr[1] := FALSE;
    ELSE
        currentOrder.generatedOrder.scorerEnabledArr[1] := TRUE;
    END_IF
END_IF
scorer1EnabledCmdOld := scorer1EnabledCmd;

IF scorer2EnabledCmd AND NOT scorer2EnabledCmdOld THEN
    IF currentOrder.generatedOrder.scorerEnabledArr[2] THEN
        currentOrder.generatedOrder.scorerEnabledArr[2] := FALSE;
    ELSE
        currentOrder.generatedOrder.scorerEnabledArr[2] := TRUE;
    END_IF
END_IF
scorer2EnabledCmdOld := scorer2EnabledCmd;

IF scorer3EnabledCmd AND NOT scorer3EnabledCmdOld THEN
    IF currentOrder.generatedOrder.scorerEnabledArr[3] THEN
        currentOrder.generatedOrder.scorerEnabledArr[3] := FALSE;
    ELSE
        currentOrder.generatedOrder.scorerEnabledArr[3] := TRUE;
    END_IF
END_IF
scorer3EnabledCmdOld := scorer3EnabledCmd;

IF scorer4EnabledCmd AND NOT scorer4EnabledCmdOld THEN
    IF currentOrder.generatedOrder.scorerEnabledArr[4] THEN
        currentOrder.generatedOrder.scorerEnabledArr[4] := FALSE;
    ELSE
        currentOrder.generatedOrder.scorerEnabledArr[4] := TRUE;
    END_IF
END_IF
scorer4EnabledCmdOld := scorer4EnabledCmd;

IF scorer5EnabledCmd AND NOT scorer5EnabledCmdOld THEN
    IF currentOrder.generatedOrder.scorerEnabledArr[5] THEN
        currentOrder.generatedOrder.scorerEnabledArr[5] := FALSE;
    ELSE
        currentOrder.generatedOrder.scorerEnabledArr[5] := TRUE;
    END_IF
END_IF
scorer5EnabledCmdOld := scorer5EnabledCmd;

IF scorer6EnabledCmd AND NOT scorer6EnabledCmdOld THEN
    IF currentOrder.generatedOrder.scorerEnabledArr[6] THEN
        currentOrder.generatedOrder.scorerEnabledArr[6] := FALSE;
    ELSE
        currentOrder.generatedOrder.scorerEnabledArr[6] := TRUE;
    END_IF
END_IF
scorer6EnabledCmdOld := scorer6EnabledCmd;

IF scorer7EnabledCmd AND NOT scorer7EnabledCmdOld THEN
    IF currentOrder.generatedOrder.scorerEnabledArr[7] THEN
        currentOrder.generatedOrder.scorerEnabledArr[7] := FALSE;
    ELSE
        currentOrder.generatedOrder.scorerEnabledArr[7] := TRUE;
    END_IF
END_IF
scorer7EnabledCmdOld := scorer7EnabledCmd;

IF scorer8EnabledCmd AND NOT scorer8EnabledCmdOld THEN
    IF currentOrder.generatedOrder.scorerEnabledArr[8] THEN
        currentOrder.generatedOrder.scorerEnabledArr[8] := FALSE;
    ELSE
        currentOrder.generatedOrder.scorerEnabledArr[8] := TRUE;
    END_IF
END_IF
scorer8EnabledCmdOld := scorer8EnabledCmd;





//-------------------------------------------------------------------------------------------------
// Detect if any knife or scorer axis is currently executing a motion command or positioning delay
//-------------------------------------------------------------------------------------------------
positioningRunning := 
    (instFB_AxisControlKnife1_Axis.commandBusy OR
    instFB_AxisControlKnife2_Axis.commandBusy OR
    instFB_AxisControlKnife3_Axis.commandBusy OR
    instFB_AxisControlKnife4_Axis.commandBusy OR
    instFB_AxisControlKnife5_Axis.commandBusy OR
    instFB_AxisControlScorer1_Axis.commandBusy OR
    instFB_AxisControlScorer2_Axis.commandBusy OR
    instFB_AxisControlScorer3_Axis.commandBusy OR
    instFB_AxisControlScorer4_Axis.commandBusy OR
    instFB_AxisControlScorer5_Axis.commandBusy OR
    instFB_AxisControlScorer6_Axis.commandBusy OR
    instFB_AxisControlScorer7_Axis.commandBusy OR  
    instFB_AxisControlScorer8_Axis.commandBusy) AND
    positioningStarted;

	
	inTargetPosition := knife1_Axis.Status.NotMoving AND
						knife2_Axis.Status.NotMoving AND
						knife3_Axis.Status.NotMoving AND
						knife4_Axis.Status.NotMoving AND
						knife5_Axis.Status.NotMoving AND						
						scorer1_Axis.Status.NotMoving AND
						scorer2_Axis.Status.NotMoving AND
						scorer3_Axis.Status.NotMoving AND	 
						scorer4_Axis.Status.NotMoving AND	 
						scorer5_Axis.Status.NotMoving AND	 
						scorer6_Axis.Status.NotMoving AND	 
						scorer7_Axis.Status.NotMoving AND	 
						scorer8_Axis.Status.NotMoving;	 
	 
	
bAllKnivesInPos := NOT positioningRunning AND
						NOT positioningStarted AND
						knife1_Axis.Status.InTargetPosition AND
						knife2_Axis.Status.InTargetPosition AND
						knife3_Axis.Status.InTargetPosition AND
						knife4_Axis.Status.InTargetPosition AND
						knife5_Axis.Status.InTargetPosition;	
						
						
//-------------------------------------------------------------------------------------------------
// Enable signal for knives: Active only if tool is enabled AND machine is cutting AND not positioning
// Home override also enables it
//-------------------------------------------------------------------------------------------------
knife1Enabled := (currentOrder.generatedOrder.knifeEnabledArr[1] AND startCutting AND NOT positioningRunning) AND NOT homeRunning AND NOT positioningStarted AND inTargetPosition;
knife2Enabled := (currentOrder.generatedOrder.knifeEnabledArr[2] AND startCutting AND NOT positioningRunning) AND NOT homeRunning AND NOT positioningStarted AND inTargetPosition;
knife3Enabled := (currentOrder.generatedOrder.knifeEnabledArr[3] AND startCutting AND NOT positioningRunning) AND NOT homeRunning AND NOT positioningStarted AND inTargetPosition;
knife4Enabled := (currentOrder.generatedOrder.knifeEnabledArr[4] AND startCutting AND NOT positioningRunning) AND NOT homeRunning AND NOT positioningStarted AND inTargetPosition;
knife5Enabled := (currentOrder.generatedOrder.knifeEnabledArr[5] AND startCutting AND NOT positioningRunning) AND NOT homeRunning AND NOT positioningStarted AND inTargetPosition;

//-------------------------------------------------------------------------------------------------
// Enable signal for scorers: Same logic as for knives
//-------------------------------------------------------------------------------------------------
scorer1Enabled := (currentOrder.generatedOrder.scorerEnabledArr[1] AND startCutting AND NOT positioningRunning) AND NOT homeRunning AND NOT positioningStarted AND inTargetPosition;
scorer2Enabled := (currentOrder.generatedOrder.scorerEnabledArr[2] AND startCutting AND NOT positioningRunning) AND NOT homeRunning AND NOT positioningStarted AND inTargetPosition;
scorer3Enabled := (currentOrder.generatedOrder.scorerEnabledArr[3] AND startCutting AND NOT positioningRunning) AND NOT homeRunning AND NOT positioningStarted AND inTargetPosition;
scorer4Enabled := (currentOrder.generatedOrder.scorerEnabledArr[4] AND startCutting AND NOT positioningRunning) AND NOT homeRunning AND NOT positioningStarted AND inTargetPosition;
scorer5Enabled := (currentOrder.generatedOrder.scorerEnabledArr[5] AND startCutting AND NOT positioningRunning) AND NOT homeRunning AND NOT positioningStarted AND inTargetPosition;
scorer6Enabled := (currentOrder.generatedOrder.scorerEnabledArr[6] AND startCutting AND NOT positioningRunning) AND NOT homeRunning AND NOT positioningStarted AND inTargetPosition;
scorer7Enabled := (currentOrder.generatedOrder.scorerEnabledArr[7] AND startCutting AND NOT positioningRunning) AND NOT homeRunning AND NOT positioningStarted AND inTargetPosition;
scorer8Enabled := (currentOrder.generatedOrder.scorerEnabledArr[8] AND startCutting AND NOT positioningRunning) AND NOT homeRunning AND NOT positioningStarted AND inTargetPosition;
END_METHOD

ACTION ACT_AlarmActive:

END_ACTION

ACTION ACT_Alarms:

END_ACTION

ACTION ACT_AuxiliaryCommands:

END_ACTION

ACTION ACT_GeneratePositions:
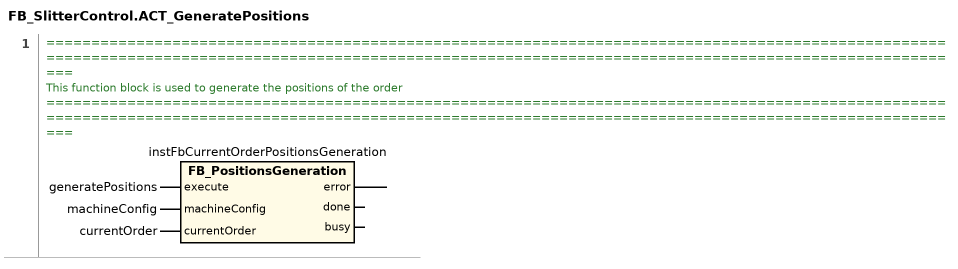
// NETWORK 1
// 					===========================================================================================================================================================================================================
//
// This function block is used to generate the positions of the order
//
// ===========================================================================================================================================================================================================
//
instFbCurrentOrderPositionsGeneration(
    execute := generatePositions,
    machineConfig := machineConfig,
    currentOrder := currentOrder); // FB_PositionsGeneration
END_ACTION

ACTION ACT_ProgramCurrentOrder:

(*==============================================================================================================================
CPNTeck - Automação industrial
(c)Copyright 2023 All Rights Reserved
_______________________________________________________________________________________________________________________________
Library: N/A 
Tested with: CX5140
Engineering: Twincat 2
Restrictions: -
Requirements: N/A
Functionality: This function is used program the current order and change the order
Support: fabio@cpnteck.com.br
Note: Parameter comments are only available in language 'English (United States)'
_______________________________________________________________________________________________________________________________
Change log table:

Version  		| Date        			| Expert in charge  	| Changes applied
01.00.01		| 29.03.2023  		| Fabio Campion            | First released version
*)


IF changeOrder AND NOT changeOrderOld THEN

	currentOrder := nextOrder;

END_IF

changeOrderOld := changeOrder;
END_ACTION

END_FUNCTION_BLOCK

// ---- Library/Machine/Slitter/FunctionBlocks/FB_KnifeSharpening.TcPOU
FUNCTION_BLOCK FB_KnifeSharpening
VAR_INPUT

	machineRunning 				: BOOL;
	manualSharpening 			: BOOL;
	measuringWheelSensor 		: BOOL;
	knifeRunningMetersReset 		: BOOL;
	knifeEnabled 				: BOOL;
	measuringWheelDiameter 		: REAL	:= 154.2;
	sharpeningSetpoint 			: REAL	:= 100.0;
	sharpeningTime				: INT 		:= 5000;

END_VAR
VAR_OUTPUT

	sharpeningSolenoid 			: BOOL;
	knifeRunningMeters 			: INT;
	knifeRunningMetersTotal 		: DINT;


END_VAR
VAR

	measuringWheelSensorOld		: BOOL;

	instSharpeningTimeTON		: TON;
	manualSharpeningOld			: BOOL;
	knifeRunningMetersResetOld	: BOOL;

END_VAR

VAR PERSISTENT

	sensorPulseCounter1 			: DINT;	(*This variable increases every pulse of the measuring wheel and resets every time the knife is shapened*)
	sensorPulseCounter2 			: DINT;	(*This variable increases every pulse of the measuring wheel and resets manualy when the knife is replaced*)


END_VAR

VAR

END_VAR

VAR CONSTANT

	PI: REAL 					:= 3.14159265359;

END_VAR


(*==============================================================================================================================
CPNTeck - Automação industrial
(c)Copyright 2022 All Rights Reserved
_______________________________________________________________________________________________________________________________
Library: N/A 
Tested with: CX5140
Engineering: Twincat 2
Restrictions: -
Requirements: N/A
Functionality: This function block is used to sharp the knifes
Support: fabio@cpnteck.com.br
Note: Parameter comments are only available in language 'English (United States)'
_______________________________________________________________________________________________________________________________
Change log table:

Version  		| Date        			| Expert in charge  	| Changes applied
01.00.01		| 18.04.2023  		| Fabio Campion            | First released version



===============================================================================================================================*)


(*Measuring wheel pulse counter*)
IF measuringWheelSensor AND NOT measuringWheelSensorOld
AND knifeEnabled  THEN

	sensorPulseCounter1 := sensorPulseCounter1 + 1;
	sensorPulseCounter2 := sensorPulseCounter2 + 1;


END_IF

measuringWheelSensorOld := measuringWheelSensor;


(*Automatic / Manual shapening*)
IF knifeRunningMeters >= sharpeningSetpoint AND machineRunning
OR  manualSharpening AND NOT manualSharpeningOld  AND machineRunning THEN

	sensorPulseCounter1 := 0; (*Reset the measuring wheel pulse counter*)
	instSharpeningTimeTON.PT := DINT_TO_TIME(SharpeningTime); (*Set the timer setpoint*)
	instSharpeningTimeTON.IN := TRUE; (*Enable the timer*)
	sharpeningSolenoid := TRUE; (*Enable the sharpening solenoid*)

END_IF

ManualSharpeningOld := ManualSharpening;

IF instSharpeningTimeTON.Q  THEN

	sharpeningSolenoid := FALSE;
	instSharpeningTimeTON.IN := FALSE;

END_IF

IF knifeRunningMetersReset AND NOT knifeRunningMetersResetOld THEN

	sensorPulseCounter2 := 0;

END_IF

knifeRunningMetersResetOld := knifeRunningMetersReset;



(*Measuring wheel meters calculation*)
KnifeRunningMeters := TRUNC_INT((sensorPulseCounter1 * (MeasuringWheelDiameter * PI)) * 0.001);
KnifeRunningMetersTotal := TRUNC_INT((sensorPulseCounter2 * (MeasuringWheelDiameter * PI)) * 0.001);



instSharpeningTimeTON();

END_FUNCTION_BLOCK

// ---- Library/Machine/Slitter/FunctionBlocks/FB_KnifeLubrification.TcPOU
FUNCTION_BLOCK FB_KnifeLubrification
VAR_INPUT

	machineRunning 				: BOOL;
	manualLubrification 			: BOOL;
	measuringWheelSensor 		: BOOL;
	knifeEnabled 				: BOOL;
	measuringWheelDiameter 		: REAL	:= 154.2;
	lubrificationSetpoint 			: REAL	:= 100.0;
	lubrificationTime				: INT 		:= 5000;

END_VAR
VAR_OUTPUT

	lubrificationSolenoid 			: BOOL;
	knifeRunningMeters 			: INT;


END_VAR
VAR

	measuringWheelSensorOld		: BOOL;
	sensorPulseCounter1 			: DINT;	(*This variable increases every pulse of the measuring wheel and resets every time the knife is shapened*)
	sensorPulseCounter2 			: DINT;	(*This variable increases every pulse of the measuring wheel and resets manualy when the knife is replaced*)

	instLubrificationTimeTON		: TON;
	manualLubrificationOld			: BOOL;
	knifeRunningMetersResetOld	: BOOL;

END_VAR
VAR

END_VAR

VAR CONSTANT

	PI: REAL 					:= 3.14159265359;

END_VAR


(*==============================================================================================================================
CPNTeck - Automação industrial
(c)Copyright 2022 All Rights Reserved
_______________________________________________________________________________________________________________________________
Library: N/A 
Tested with: CX5140
Engineering: Twincat 2
Restrictions: -
Requirements: N/A
Functionality: This function block is used to lubrificate the knifes in the disired interval.
Support: fabio@cpnteck.com.br
Note: Parameter comments are only available in language 'English (United States)'
_______________________________________________________________________________________________________________________________
Change log table:

Version  		| Date        			| Expert in charge  	| Changes applied
01.00.01		| 18.04.2023  		| Fabio Campion            | First released version



===============================================================================================================================*)


(*Measuring wheel pulse counter*)
IF measuringWheelSensor AND NOT measuringWheelSensorOld
AND knifeEnabled  THEN

	sensorPulseCounter1 := sensorPulseCounter1 + 1;
	sensorPulseCounter2 := sensorPulseCounter2 + 1;


END_IF

measuringWheelSensorOld := measuringWheelSensor;


(*Automatic / Manual shapening*)
IF knifeRunningMeters >= lubrificationSetpoint AND machineRunning
OR  manualLubrification AND NOT manualLubrificationOld  AND machineRunning THEN

	sensorPulseCounter1 := 0; (*Reset the measuring wheel pulse counter*)
	instLubrificationTimeTON.PT := DINT_TO_TIME(LubrificationTime); (*Set the timer setpoint*)
	instLubrificationTimeTON.IN := TRUE; (*Enable the timer*)
	lubrificationSolenoid := TRUE; (*Enable the sharpening solenoid*)

END_IF

ManualLubrificationOld := ManualLubrification;

IF instLubrificationTimeTON.Q  THEN

	lubrificationSolenoid := FALSE;
	instLubrificationTimeTON.IN := FALSE;

END_IF


(*Measuring wheel meters calculation*)
KnifeRunningMeters := TRUNC_INT((sensorPulseCounter1 * (MeasuringWheelDiameter * PI)) * 0.001);

instLubrificationTimeTON();

END_FUNCTION_BLOCK

// ---- Library/AxisControl/FB_SimpleAxisControl.TcPOU
FUNCTION_BLOCK FB_SimpleAxisControl
VAR_INPUT

	enable							: BOOL   := FALSE;		(* TRUE: Enable functionality of FB *)
	enableAxis						: BOOL   := FALSE;		(* TRUE: Set axis enable; FALSE: Remove axis enable *)
	resetAxis						: BOOL   := FALSE;		(* Rising edge: Acknowledgement of technology alarms or restart of the axis (depending on configuration) *)
	jogForward						: BOOL   := FALSE;		(* Rising edge: Move an axis in jog mode (forward); Falling edge: Stop jogging *)
	jogBackward						: BOOL   := FALSE;	          (* Rising edge: Move an axis in jog mode (backward); Falling edge: Stop jogging *)
	moveVelocity					: BOOL   := FALSE;	          (* Rising edge: Move an axis at constant velocity/speed *)
	stop							: BOOL   := FALSE;	          (* Rising edge: Brake an axis until it comes to a standstill *)
	fastStop						: BOOL   := FALSE;	          (* Rising edge: Brake an axis until it comes to a standstill (with fastStop dynamics) *)
	torqueLimiting					: BOOL   := FALSE;	          (* TRUE: Enable force/torque limiting *)
	homing							: BOOL   := FALSE;	          (* Rising edge: Home axis *)
	homingSensor					: BOOL   := FALSE;	          (* Rising edge: Home sensor input singnal *)
	posRelative						: BOOL   := FALSE;	          (* Rising edge: Move an axis relative to its position when execution of the job began *)
	posAbsolute						: BOOL   := FALSE;	          (* Rising edge: Move an axis to an absolute position *)
	posSuperimposed					: BOOL   := FALSE;	          (* Rising edge: Start a superimposed positioning *)
	gearInRelative					: BOOL   := FALSE;	          (* Rising edge: Start a gearing operation (relative) *)
	gearInAbsolute					: BOOL   := FALSE;	          (* Rising edge: Start a gearing operation (absolute) *)
	camIn							: BOOL   := FALSE;	          (* Rising edge: Start a camming operation *)
	phasing							: BOOL   := FALSE;	          (* Rising edge: Start a phasing operation *)

END_VAR

VAR_OUTPUT

	valid							: BOOL   := FALSE;	          (* TRUE: Valid set of output values available at the FB *)
	busy							: BOOL   := FALSE;	          (* TRUE: FB is working and new output values can be expected *)
	error							: BOOL   := FALSE;	          (* TRUE: An error occurred while processing the FB *)
	status							: WORD   := STATUS_NO_CALL;	 (* Current status of FB *)
	axisEnabled						: BOOL   := FALSE;	          (* TRUE: The technology object is enabled. Motion commands can be executed *)
	resetActive						: BOOL   := FALSE;	          (* TRUE: Reset/Restart of the axis is active *)
	commandBusy						: BOOL   := FALSE;	          (* TRUE: The selected basic motion command is being executed *)
	commandDone						: BOOL   := FALSE;	          (* TRUE: The selected basic motion command has completed without error *)
	commandAborted					: BOOL   := FALSE;	          (* TRUE: The selected basic motion command has been aborted *)
	inVelocity						: BOOL   := FALSE;	          (* TRUE: The setpoint velocity/speed was reached and will be maintained *)
	inLimitation					: BOOL   := FALSE;	          (* TRUE: The drive is operating at the force/torque limit *)
	homingCommandBusy				: BOOL   := FALSE;	          (* TRUE: Homing command is being executed *)
	homingCommandDone				: BOOL   := FALSE;	          (* TRUE: Homing command has completed without error *)
	homingCommandAborted			: BOOL   := FALSE;	          (* TRUE: Homing command has been aborted *)
	superimposedBusy				: BOOL   := FALSE;	          (* TRUE: The selected superimposed motion command is being executed *)
	superimposedDone				: BOOL   := FALSE;	          (* TRUE: The selected superimposed motion command  has completed without error *)
	superimposedAborted				: BOOL   := FALSE;	          (* TRUE: The selected superimposed motion command has been aborted *)
	inClamping						: BOOL   := FALSE;	          (* TRUE: The drive is kept at the fixed stop (clamping), the axis position is within the positioning tolerance *)
	startSync						: BOOL   := FALSE;	          (* TRUE: The axis is synchronizing to the leading axis *)
	inSync							: BOOL   := FALSE;	          (* TRUE: The axis is synchronized to the leading axis *)
	inSimulation					: BOOL   := FALSE;	          (* TRUE: Synchronous operation is being simulated *)
	jogSelected						: BOOL   := FALSE;	          (* TRUE: Jogging is active *)
	moveVelocitySelected			: BOOL   := FALSE;	          (* TRUE: Moving with constant velocity/speed is active *)
	stopSelected					: BOOL   := FALSE;	          (* TRUE: Stopping is active *)
	fastStopSelected				: BOOL   := FALSE;	          (* TRUE: Stopping is active (with fastStop dynamics) *)
	torqueLimitingSelected			: BOOL   := FALSE;	          (* TRUE: Force/Torque limiting is active *)
	homingSelected					: BOOL   := FALSE;	          (* TRUE: Homing is active *)
	posRelativeSelected				: BOOL   := FALSE;	          (* TRUE: Relative positioning is active *)
	posAbsoluteSelected				: BOOL   := FALSE;	          (* TRUE: Absolute positioning is active *)
	posSuperimposedSelected			: BOOL   := FALSE;	          (* TRUE: Superimposed positioning is active *)
	gearInRelativeSelected			: BOOL   := FALSE;	          (* TRUE: Relative gearing is active *)
	gearInAbsoluteSelected			: BOOL   := FALSE;	          (* TRUE: Absolute gearing is active *)
	camInSelected					: BOOL   := FALSE;	          (* TRUE: Camming is active *)
	phasingSelected					: BOOL   := FALSE;	          (* TRUE: Phasing is active *)
	diagnostics						: LAxisCtrl_typeDiagnostics;	(* Diagnostics structure *)

END_VAR

VAR_IN_OUT

	axis							: AXIS_REF;		  (* Reference to axis to be controlled *)
	master							: AXIS_REF;		  (* Reference to leading axis for synchronous motion *)
	configuration					: LAxisCtrl_typeAxisConfig;	 (* Structure for parameters *)

END_VAR

VAR
	statErrorUserCleared			: BOOL   := FALSE;	          (* Error occurred that can only be solved by user; rising edge at enable input necessary *)
	statErrorAutoCleared			: BOOL   := FALSE;	          (* Error occurred that can be acknowledged by FB *)
	statStatus						: WORD   := STATUS_NO_CALL;	 (* Internal variable for status *)
	statDiagnostics					: LAxisCtrl_typeDiagnostics;	(* Internal variable for diagnostics *)
	statEnableOld					: BOOL   := FALSE;	          (* Old value of enable for edge detection *)
	statFBState						: SINT   := AXIS_MOTION;	    (* State of FB (function block state machine) *)
	statFirstCycleReset				: BOOL   := TRUE;	           (* TRUE: First cycle of reset command *)
	statPowerErrorOld				: BOOL   := FALSE;	          (* Old value of MC_Power.error *)
	statResetState					: INT    := CMD_IDLE;	       (* State of reset command *)
	statFirstCycleResetError		: BOOL   := FALSE;	          (* TRUE: First cycle of error in reset command *)
	statExtendedCommand				: DWORD  := CMD_NO_SELECTION;              (* Variable for requested extended command (e.g. resetAxis, torquelimiting, homing) *)
	statExtendedCommandOld			: DWORD  := CMD_NO_SELECTION;              (* Old value of variable for requested extended command *)
	statEnableAxisOld				: BOOL   := FALSE;	          (* Old value of enableAxis for edge detection *)
	statEmptyDiagnostics			: LAxisCtrl_typeDiagnostics;	(* Internal empty diagnostic structure *)
	statHomingOld					: BOOL   := FALSE;	          (* Old value of variable for homing command input *)
	statFirstCycleHoming			: BOOL   := TRUE;	           (* TRUE: First cycle in homing command *)
	statPassiveHomingState			: DINT   := NO_HOMING_ACTIVE;              (* Current selected passive homing mode *)
	statExeOfHoming					: INT    := CMD_BUSY;	       (* Current state of execution of homing command *)
	statBasicCommand				: DWORD  := CMD_NO_SELECTION;              (* Variable for requested basic motion command *)
	statBasicCommandOld				: DWORD  := CMD_NO_SELECTION;              (* Old value of variable for requested basic motion command *)
	statBasicMotionState			: DINT   := NO_SELECTION;	   (* State of selected basic motion command *)
	statExeOfBasicMotion			: INT    := CMD_BUSY;	       (* State of execution of current state of basic motion *)
	statFirstCycleBasicMotion		: BOOL   := TRUE;	           (* TRUE: First cycle in respective state fo basic motion functionality *)
	statApplicativeBasicMotionError	: BOOL   := FALSE;	          (* TRUE: applicative error occurred (e.g. invalid direction configured) *)
	statVelocityChangeOnTheFly		: BOOL   := FALSE;	          (* Velocity change on the fly is active *)
	statVelocity					: LREAL  := 0.0;	            (* Internal variable for velocity *)
	statAcceleration				: LREAL  := 0.0;	            (* Internal variable for acceleration *)
	statAbortAcceleration			: BOOL   := FALSE;	          (* FALSE: The current acceleration at the start of the job is reduced using the configured jerk. Afterwards, the deceleration builds up; TRUE: The acceleration is set to 0.0 at the start of the job, and the deceleration immediately builds up. *)
	statDeceleration				: LREAL  := 0.0;	            (* Internal variable for deceleration *)
	statJerk						: LREAL  := 0.0;	            (* Internal variable for jerk *)
	statPositionControlled			: BOOL   := TRUE;	           (* FALSE: Non position-controlled operation; TRUE: Position-controlled operation *)
	statFirstCycleDone				: BOOL   := FALSE;	          (* TRUE: First cycle of done at fastStop *)
	statTorqueLimitingState			: SINT   := NO_TORQUE_LIMITING_ACTIVE;     (* Current executed state for torquelimiting functionality *)
	statTorqueLimitingErrorOld		: BOOL   := FALSE;	          (* TRUE: Error at Torquelimiting occurred last cycle *)
	statTorqueLimit					: LREAL  := -1.0;	           (* Value of force/torque limiting (in the configured unit of measurement) *)
	statJogMode						: DINT   := JOG_MODE_CONTINUOUS;           (* Current selected jog mode *)
	statDirection					: INT    := SPECIFIED_DIR;	  (* Internal variable for direction of rotation of the axis *)
	statHomingPosition				: LREAL  := 0.0;	            (* The specified value is used according to the selected "Mode". *)
	statHomingSubState				: SINT   := HOMING_IDLE;	    (* Current subState of execution of homing functionality *)
	statIncJogSubState				: SINT   := INC_JOG_IDLE;	   (* Current subState of execution of jog incremental functionality *)
	statIncJogStartPosition			: LREAL  := 0.0;	            (* Last stored axis position (for incremental jogging) *)
	statIncJogDirectionOld			: INT    := 0;	              (* Old value of direction of executing incremental jogging *)
	statIncrement					: LREAL  := 0.0;	            (* Jog Incremental: distance of Increment (positive or negative) *)
	statIncJogDistance				: LREAL  := 0.0;	            (* Jog Incremental: current distance to destination position *)
	statResetIncJog					: BOOL   := TRUE;	           (* TRUE: First cycle in incremental jogging state (detection of new increment) *)
	statPosition					: LREAL  := 0.0;	            (* Internal variable for position *)
	statPositionChangeOnTheFly		: BOOL   := FALSE;	          (* Position change on the fly is active *)
	statHomingMode					: INT    := DIRECT_HOMING;	  (* Operating Mode of MC_HOME command *)
	statActiveHomingState			: DINT   := NO_HOMING_ACTIVE;              (* Current selected active homing mode *)
	statSupImpCommand				: DWORD  := CMD_NO_SELECTION;              (* Variable for requested superimposed motion command *)
	statSupImpCommandOld			: DWORD  := CMD_NO_SELECTION;              (* Old value of variable for requested superimposed motion command *)
	statSupImpMotionState	        : DINT   := NO_SELECTION;	   (* Current selected superimposed motion functionality *)
	statExeOfSupImpMotionState		: INT    := CMD_BUSY;	       (* Current state of execution of superimposed basic motion *)
	statFirstCycleSupImpMotion			: BOOL   := TRUE;	           (* TRUE: First cycle in positioning (superimposed) functionality *)
	statSupImpMotionPosition			: LREAL  := 0.0;	            (* Position setpoint (for posSuperimposed command) *)
	statApplicativeSupImpMotionError		: BOOL   := FALSE;	          (* TRUE: applicative error occurred (e.g. invalid direction configured) *)
	statRatioChangeOnTheFly			: BOOL   := FALSE;	          (* Ratio change on the fly is active *)
	statChangePhaseShiftOnTheFly	: BOOL   := FALSE;	          (* Phase shift change on the fly is active *)
	statPhaseShift					: LREAL  := 0.0;	            (* Relative/Absolute master value shift *)
	statPhaseAbsolute				: BOOL   := TRUE;	           (* Indicates the type of phase shift (TRUE: The phase shift is taken over as an absolute value; FALSE: The phase shift is added to an existing offset) *)
	statRatioNumerator				: DINT   := 1;	              (* Gear ratio numerator *)
	statRatioDenominator			: DINT   := 1;	              (* Gear ratio denominator *)
	statEnableAxis					: BOOL   := FALSE;	          (* Internal variable for enabling axis *)
	statSyncMotionSimulationState	: SINT   := AXIS_NOT_IN_SIM;	(* Current executed state for synchronized motion simulation *)
	statSynchronizedMotionErrorOld	: BOOL   := FALSE;	          (* Old value of MC_SynchronizedMotionSimulation.error *)
	statMainSelectionState			: INT    := 0;	              (* Current executed State for execution of basic motion commands or reset of waiting gearing / camming commands *)
	statMasterSyncPosition			: LREAL  := 0.0;	            (* Synchronous position of leading axis. Position of the following axis starting from which the leading and following axes move synchronously *)
	statSlaveSyncPosition			: LREAL  := 0.0;	            (* Synchronous position of leading axis. Position of the leading axis starting from which the leading and following axes move synchronously *)
	statSyncDirection				: DINT   := FORWARD_DIR;	    (* Direction of synchronization *)
	statMasterStartDistance			: LREAL  := 0.0;	            (* Master value distance (when "SyncProfileReference" = 1) *)
	statSyncProfileReference		: DINT   := 0;	              (* Type of synchronization *)
	statApplicationMode				: DINT   := 0;	              (* Application of cam *)

	instPower						: MC_Power;		  (* Instance of MC_Power *)
	instReset						: MC_Reset;		  (* Instance of MC_Reset *)
	instHome						: MC_Home;		   (* Instance of MC_Home *)
	instHalt						: MC_Halt;		   (* Instance of MC_Halt *)
	instMoveJog						: MC_Jog;		    (* Instance of MC_MoveJog *)
	instTorqueLimiting				: MC_TORQUELIMITING;	        (* Instance of MC_TorqueLimiting *)
	instMoveVelocity				: MC_MoveVelocity;	          (* Instance of MC_MoveVelocity *)
	instMoveRelative				: MC_MoveRelative;	          (* Instance of MC_MoveRelative *)
	instMoveAbsolute				: MC_MoveAbsolute;	          (* Instance of MC_MoveAbsolute *)
	instMoveSuperimposed			: MC_MoveSuperImposed;	      (* Instance of MC_MoveSuperimposed *)
	instGearIn						: MC_GearIn;		 (* Instance of MC_GearIn *)
	instPhasingAbsolute				: MC_PhasingAbsolute;	       (* Instance of MC_PhasingAbsolute *)
	instPhasingRelative				: MC_PhasingRelative;	       (* Instance of MC_PhasingRelative *)
	instGearInPos					: MC_GearInDyn;	             (* Instance of MC_GearInPos *)
//	instCamIn						: MC_CamIn;		  (* Instance of MC_CamIn *)
	instSyncMotionSimulation		: MC_SYNCHRONIZEDMOTIONSIMULATION;         (* Instance of MC_SynchronizedMotionSimulation *)
	instTimerTON					: TON;
	StatusWord						: INT;

END_VAR

VAR

	tempNewExtendedCmd				: DINT;		      (* Temporary variable for extended command *)
	tempEnableAxis					: BOOL;		      (* Temporary variable for enableAxis *)
	tempErrorInCmd					: BOOL;		      (* Temporary variable for error in actual command *)
	tempRisingCmd					: DWORD;		     (* Temporary DWord which indicates all rising edges of command word *)
	tempStopCmdSelected				: BOOL;		      (* TRUE: Stop or faststop selected in current cycle *)
	tempDword						: DWORD;		     (* Temporary DWord for evaluation of rising edges of basic command word *)
	tempIndex						: INT;		       (* Temporary index *)
	tempCountRisEdges				: USINT;		     (* Temporary counter for rising edges in command word *)
	tempNewBasicMotionCmd			: DINT;		      (* Temporary variable for basic motion command *)
	tempStateChangeActive			: BOOL;		      (* TRUE: State change is active, stay in loop for one more cycle *)
	tempStatusWord					: DWORD;		     (* Temporary variable for statusword of axis *)
	tempNewSupImpCmd				: DINT;		      (* Temporary variable for superimposed motion command *)
	tempHoming						: BOOL;		      (* Temporary variable for homing command *)
	tempFalse						: BOOL;

END_VAR

VAR CONSTANT

	AXIS_MOTION								: SINT   := 1;	              (* State of FB: MotionState, new commands are evaluated *)
	FB_ERROR								: SINT   := 5;	              (* State of FB: Error, falling edge at FB_ENABLE required *)
	CMD_NO_SELECTION						: DWORD  := 16#0000_0000;	   (* No command is selected *)
	NO_SELECTION							: INT    := 0;	              (* State of basicMotion/superimposedMotion: No execution of a command *)
	AXIS_FAST_STOPPING						: SINT   := 2;	              (* State of FB: StoppingState, MC_HALT is executed, new commands are not evaluated *)
	AXIS_STOP_ON_ERROR_SELECTION			: SINT   := 3;	              (* State of FB: ErrorState: Selection if StopOnError must be executed (depending on configuration) *)
	AXIS_STOP_ON_ERROR_EXECUTION			: SINT   := 4;	              (* State of FB: ErrorState: Execution of StopOnError *)
	FAST_STOP_SELECTED						: INT    := 1;	              (* State of basicMotion: Execution of fast stop command *)
	STOP_SELECTED							: INT    := 2;	              (* State of basicMotion: Execution of stop command *)
	JOG_FORWARD_SELECTED					: INT    := 4;	              (* State of basicMotion: Execution of jog forward command *)
	JOG_BACKWARD_SELECTED					: INT    := 8;	              (* State of basicMotion: Execution of jog backward command *)
	JOG_FW_AND_BW_SELECTED					: INT    := 12;	             (* State of basicMotion: Execution of jog command if forward and backward are selected *)
	MOVE_VELOCITY_SELECTED					: INT    := 16;	             (* State of basicMotion: Execution of move velocity command *)
	ACTIVE_HOMING_SELECTED					: INT    := 1024;	           (* State of basicMotion: Execution of active homing command *)
	POS_RELATIVE_SELECTED					: INT    := 32;	             (* State of basicMotion: Execution of position command (relative) *)
	POS_ABSOLUTE_SELECTED					: INT    := 64;	             (* State of basicMotion: Execution of position command (absolute) *)
	GEAR_IN_RELATIVE_SELECTED				: INT    := 128;	            (* State of basicMotion: Execution of gearIn command *)
	GEAR_IN_ABSOLUTE_SELECTED				: INT    := 256;	            (* State of basicMotion: Execution of gearInPos command *)
	CAM_IN_SELECTED							: INT    := 512;	            (* State of basicMotion: Execution of camIn command *)
	POS_SUPERIMPOSED_SELECTED				: INT    := 1;	              (* State of superimposedMotion: Execution of posSuperimposed command *)
	PHASING_SELECTED							: INT    := 2;	              (* State of superimposedMotion: Execution of phasing command *)
	CMD_IDLE									: INT    := 0;	              (* State of basicMotion command: No execution *)
	CMD_BUSY								: INT 	   := 1;	              (* State of basicMotion command: Subsequent call *)
	CMD_DONE								: INT 	   := 2;	              (* State of basicMotion command: Finished with "DONE" *)
	CMD_ABORTED								: INT    := 4;	              (* State of basicMotion command: Finished with "ABORTED" *)
	CMD_ERROR								: INT    := 8;	              (* State of basicMotion command: Finished with "ERROR" *)
	CMD_END_PROCESS							: INT    := 16;	             (* State of basicMotion command: Finished with other reason *)
	JOG_MODE_CONTINUOUS						: INT    := 0;	              (* Jogmode continuous selected (MC_MOVEJOG) *)
	NO_TORQUE_LIMITING_ACTIVE				: SINT   := 0;	              (* State of torquelimiting command: Not enabled *)
	TORQUE_LIMTING_SELECTED					: SINT   := 1;	              (* State of torquelimiting command: Torquelimiting is active *)
	TORQUE_LIMITING_DISABLE					: SINT   := 10;	             (* State of torquelimiting command: Torquelimiting is disabling *)
	BITPOSITION_BASIC_MOTION_CMD			: SINT   := 4;	              (* First bitposition for detecting rising edges at basic motion command word *)
	BIT_POS_LAST								: SINT   := 15;	             (* Last bitposition for detecting rising edges at command word *)
	SPECIFIED_DIR								: INT    := 0;	              (* The sign of the velocity specified at the "Velocity" parameter defines the direction of rotation. *)
	NO_HOMING_ACTIVE							: SINT   := -10;	            (* State of homing command: No homing active *)
	STANDARD_HOMING							: SINT   := -1;	             (* State of homing command: (Standard) homing with MC_HOME *)
	BITPOSITION_SUPERIMPOSED_MOTION_CMD           	: SINT   := 0;	              (* First bitposition for detecting rising edges at superimposed motion command word *)
	FIXED_STOP_DETECTION_ACTIVE				: SINT   := 2;	              (* State of torquelimiting command: Homing on fixed stop is active *)
	FIXED_STOP_DETECTION_FINISHED				: SINT   := 3;	              (* State of torquelimiting command: Homing on fixed stop is finished *)
	AUTOMATIC_MODE_CHANGE					: SINT   := 4;	              (* State of torquelimiting command: automatic mode change is active (form 1 to 0) *)
	FIXED_STOP_DETECTION_ERROR_IN_CLAMPING		: SINT   := 5;	              (* State of torquelimiting command: Error occurred at homing on fixed stop process, axis is in clamping *)
	FIXED_STOP_DETECTION_ERROR_NOT_IN_CLAMPING	: SINT   := 6;	              (* State of torquelimiting command: Error occurred at homing on fixed stop process, axis is not in clamping *)
	HOMING_ON_FIXED_STOP						: SINT   := 0;	              (* State of homing command: Applicative homing on fixed stop process active *)
	MODE_FIXED_STOP_DETECTION					: INT    := 1;	              (* Fixed stop detection (Mode for MC_TORQUELIMITING) *)
	FORWARD_DIR								: INT    := 1;	              (* Positive/Forward direction of rotation *)
	BACKWARD_DIR								: INT    := 2;	              (* Negative/Backward direction of rotation *)
	SHORTEST_WAY_DIR							: INT    := 3;	              (* Shortest path *)
	DIRECT_HOMING							: INT    := 0;	              (* Direct homing (absolute). Parameter "position" at MC_HOME is effective *)
	ACTIVE_HOMING							: INT    := 3;	              (* Active homing. Parameter "position" at MC_HOME is effective *)
	ACTIVE_HOMING_TO_DEF_VALUE				: INT    := 5;	              (* Active homing. The configured home position value in technology object is effective *)
	ABSOLUTE_ENCODER_ADJUSTMENT				: INT    := 7;	              (* Absolute encoder adjustment (absolute) *)
	INCREMENTAL_ENCODER						: INT    := 0;	              (* Encodertype INCREMENTAL *)
	HOMING_IDLE								: SINT   := 0;	              (* SubState of homing on fixed stop process: Idle *)
	HOMING_FIXED_STOP_DETECTION				: SINT   := 1;	              (* SubState of homing on fixed stop process: Detecting fixed stop *)
	HOMING_PROCESS							: SINT   := 2;	              (* SubState of homing on fixed stop process: Homeprocess (MC_HOME) *)
	HOMING_POSITION							: SINT   := 3;	              (* SubState of homing on fixed stop process: Positioning to homeposition *)
	INC_JOG_IDLE								: SINT   := 0;	              (* Substate of incremental jog process: Idle *)
	INC_JOG_START							: SINT   := 1;	              (* Substate of incremental jog process: Start moving *)
	INC_JOG_STOP								: SINT   := 3;	              (* Substate of incremental jog process: Stop moving *)
	JOG_MODE_NEW_INCREMENT					: INT    := 1;	              (* Jogmode incremental selected - start always with new increment when command is selected *)
	JOG_MODE_CONTINUE_INCREMENT				: INT    := 2;	              (* Jogmode incremental selected - continue with increment when command is selected again *)
	APPLICATION_MODE_ONCE					: INT    := 0;	              (* Application of the cam: Once/not cyclic (MC_CAMIN) *)
	CALL_BASIC_MOTION							: INT    := 0;	              (* State of MainSelectionState: Regular execution of basic motion commands *)
	RESET_GEARING							: INT    := 1;	              (* State of MainSelectionState:Reset of waiting synchronous commands *)
	AXIS_NOT_IN_SIM							: SINT   := 0;	              (* State of motionSimulation: Axis is not in simulation *)
	AXIS_STATE_SET_SIM						: SINT   := 1;	              (* State of motionSimulation: Setting axis in simulation *)
	AXIS_DISABLE								: SINT   := 2;	              (* State of motionSimulation: Disable axis *)
	AXIS_STATE_IN_SIM							: SINT   := 3;	              (* State of motionSimulation: Axis is in simulation *)
	AXIS_ENABLE								: SINT   := 4;	              (* State of motionSimulation: Enable axis *)
	AXIS_STATE_RESET_SIM						: SINT   := 5;	              (* State of motionSimulation: Resetting axis simulation *)
	STATUS_NO_CALL							: WORD   := 16#7000;	        (* No call of FB *)
	STATUS_FB_FIRST_CALL						: WORD   := 16#7001;	        (* First cycle of FB after enabling *)
	STATUS_SUBSEQUENT_CALL					: WORD   := 16#7002;	        (* FB enabled *)
	ERR_INVALID_BASIC_MOTION_CMD				: WORD   := 16#8001;	        (* Invalid basic command selected (rising edge at 2 or more basic motion command inputs) *)
	ERR_INVALID_EXTENDED_CMD					: WORD   := 16#8002;	        (* Invalid extended command selected (rising edge at torque limiting and homing on fixed stop) *)
	ERR_INVALID_SUPERIMPOSED_MOTION_CMD		: WORD   := 16#8003;	        (* Invalid superimposed command selected (rising edge at 2 or more superimposed motion command inputs) *)
	ERR_INVALID_CAM							: WORD   := 16#8200;	        (* Error occurred during camIn command (invalid cam connected at cam input) *)
	ERR_INVALID_JOG_MODE						: WORD   := 16#8201;	        (* Invalid jog mode selected *)
	ERR_INVALID_HOMING_EXTENDED_MODE			: WORD   := 16#8202;	        (* Command Error: Invalid extended homing mode selected *)
	ERR_TORQUE_LIMITING_NOT_ALLOWED			: WORD   := 16#8203;	        (* Error during extended homing command - torque limiting not allowed during homing on fixed stop is active or axis in clamping *)
	ERR_INVALID_JOG_DIR						: WORD   := 16#8204;	        (* Invalid direction selected (jog forward and jog backward) *)
	ERR_INVALID_POS_RELATIVE_DIR				: WORD   := 16#8205;	        (* Invalid direction is set for relative positioning command *)
	ERR_INVALID_POS_SUPERIMPOSED_DIR			: WORD   := 16#8206;	        (* Invalid direction is set for superimposed positioning command *)
	ERR_HOMING_MODE_NOT_ALLOWED				: WORD   := 16#8207;	        (* Passive/Direct homing is not allowed during extended homing mode (homing on fixed stop process) is active *)
	ERR_MODULO_NOT_ALLOWED					: WORD   := 16#8208;	        (* Extended homing mode (homing on fixed stop process) is not allowed with modulo axis *)
	ERR_INVALID_TORQUE_LIMIT					: WORD   := 16#8209;	        (* Configured torque limit value for extended homing mode (homing on fixed stop process)     = 0 *)
	ERR_INVALID_VELOCITY						: WORD   := 16#820A;	        (* Configured velocity (in technology object) for active homing		= 0 *)
	ERR_MC_POWER							: WORD   := 16#8600;	        (* Error occurred during MC_POWER command *)
	ERR_MC_RESET							: WORD   := 16#8601;	        (* Error occurred during MC_RESET command *)
	ERR_MC_HOME								: WORD   := 16#8602;	        (* Error occurred during MC_HOME command *)
	ERR_MC_TORQUELIMITING						: WORD   := 16#8603;	        (* Error occurred during MC_TORQUELIMITING command *)
	ERR_MC_HALT								: WORD   := 16#8604;	        (* Error occurred during MC_HALT command *)
	ERR_MC_MOVEJOG							: WORD   := 16#8605;	        (* Error occurred during MC_MOVEJOG command (continuous jogging) *)
	ERR_MC_MOVEVELOCITY						: WORD   := 16#8606;	        (* Error occurred during MC_MOVEVELOCITY command *)
	ERR_MC_MOVERELATIVE						: WORD   := 16#8607;	        (* Error occurred during MC_MOVERELATIVE command *)
	ERR_MC_MOVEABSOLUTE						: WORD   := 16#8608;	        (* Error occurred during MC_MOVEABSOLUTE command *)
	ERR_MC_MOVESUPERIMPOSED					: WORD   := 16#8609;	        (* Error occurred during MC_MOVESUPERIMPOSED command *)
	ERR_MC_GEARIN							: WORD   := 16#860A;	        (* Error occurred during MC_GEARIN command *)
	ERR_MC_PHASINGABSOLUTE					: WORD   := 16#860B;	        (* Error occurred during MC_PHASINGABSOLUTE command *)
	ERR_MC_PHASINGRELATIVE					: WORD   := 16#860C;	        (* Error occurred during MC_PHASINGRELATIVE command *)
	ERR_MC_CAMIN								: WORD   := 16#860D;	        (* Error occurred during MC_CAMIN command *)
	ERR_MC_GEARINPOS							: WORD   := 16#860E;	        (* Error occurred during MC_GEARINPOS command *)
	ERR_MC_SYNCHRONIZEDMOTIONSIMULATION		: WORD   := 16#860F;	        (* Error occurred during MC_SYNCHRONIZEDMOTIONSIMULATION command *)
	ERR_UNDEFINED_FB_STATE					: WORD   := 16#8700;	        (* Error due to an undefined FB state *)
	ERR_UNDEFINED_RESET_STATE				: WORD   := 16#8701;	        (* Error due to an undefined reset state *)
	ERR_UNDEFINED_BASIC_MOTION_STATE			: WORD   := 16#8702;	        (* Error due to an undefined basic motion state *)
	ERR_UNDEFINED_TORQUE_LIMITING_STATE		: WORD   := 16#8703;	        (* Error due to an undefined torque limiting state *)
	ERR_UNDEFINED_INCREMENTAL_JOG_STATE		: WORD   := 16#8704;	        (* Error due to an undefined incremental jog state *)
	ERR_UNDEFINED_INCREMENTAL_JOG_SUBSTATE	: WORD   := 16#8705;	        (* Error due to an undefined incremental jog substate *)
	ERR_UNDEFINED_EXTENDED_HOMING_STATE		: WORD   := 16#8706;	        (* Error due to an undefined homing state *)
	ERR_UNDEFINED_EXTENDED_HOMING_SUBSTATE	: WORD   := 16#8707;	        (* Error due to an undefined homing substate *)
	ERR_UNDEFINED_SUPERIMPOSED_MOTION_STATE	: WORD   := 16#8708;	        (* Error due to an undefined superimposed motion state *)
	ERR_UNDEFINED_MOTION_SIMULATION_STATE		: WORD   := 16#8709;	        (* Error due to an undefined synchronized motion simulation state *)
	ERR_UNDEFINED_MAIN_SELECTION_STATE		: WORD   := 16#870A;	        (* Error due to an undefined main selection state *)

END_VAR


(*================================================================================
CPNTeck - Automação ind.
(c)Copyright 2022 All Rights Reserved
_______________________________________________________________________________________________________________________________
Library: N/A 
Tested with: CX5140
Engineering: Twincat 3
Restrictions: -
Requirements: N/A
Functionality: This function block offers basic functionalities for axis control
Support: fabio@cpnteck.com.br
Note: Parameter comments are only available in language 'English (United States)'
_______________________________________________________________________________________________________________________________
Change log table:
Version  		| Date        		| Expert in charge  		| Changes applied

01.00.01		| 12.10.2016  		| Fabio Campion                | First released version



================================================================================*)



(*----------------------------------------------------------------------------------------------*)
(* Enable / disable FB									*)
(*----------------------------------------------------------------------------------------------*)

{REGION "ENABLE_FB"}
IF NOT enable AND statEnableOld THEN
    {REGION "FALLING_EDGE_AT_ENABLE_FB"}

    (* Reset outputs									   *)
    (*==========================================================*)
    (* Error and valid outputs are reset with falling edge of enable input	   *)
	
    error  := FALSE;
    valid  := FALSE;
    status := STATUS_NO_CALL;


   (* Reset status outputs *)
    axisEnabled := FALSE;
    resetActive := FALSE;

   (* Reset outputs for homing commands *)
    homingCommandBusy := FALSE;
    homingCommandDone := FALSE;
    homingCommandAborted := FALSE;
    homingSelected := FALSE;

   (* Reset outputs for torquelimiting command *)
    torqueLimitingSelected := FALSE;
    inLimitation           := FALSE;

   (* Reset outputs for basic motion commands *)
    commandDone := FALSE;
    commandBusy := FALSE;
    commandAborted := FALSE;
    inVelocity := FALSE;
    fastStopSelected := FALSE;
    stopSelected := FALSE;
    jogSelected := FALSE;
    moveVelocitySelected := FALSE;
   (* Outputs for for up to LAxisCtrl_PosAxis *)
    posRelativeSelected := FALSE;
    posAbsoluteSelected := FALSE;
    inClamping := FALSE;

   (* Reset outputs for superimposed motion commands *)
    superimposedBusy := FALSE;
    superimposedDone := FALSE;
    superimposedAborted := FALSE;
    posSuperimposedSelected := FALSE;
    startSync := FALSE;
    inSync := FALSE;
    gearInRelativeSelected := FALSE;
    inSimulation := FALSE;
    gearInAbsoluteSelected := FALSE;
    phasingSelected := FALSE;
    camInSelected := FALSE;

    (* Reset internal variables								   *)
    (*==========================================================*)


    statErrorUserCleared := FALSE;
    statErrorAutoCleared := FALSE;
    statStatus := STATUS_NO_CALL;
    statDiagnostics := statEmptyDiagnostics;

    statFBState := AXIS_MOTION;
    statFirstCycleReset := FALSE;
    statPowerErrorOld := FALSE;
    statResetState := CMD_IDLE;
    statFirstCycleResetError := FALSE;

    statExtendedCommand := CMD_NO_SELECTION;
    statExtendedCommandOld := CMD_NO_SELECTION;
    statEnableAxisOld := FALSE;
    statHomingOld := FALSE;
    statFirstCycleHoming := FALSE;
    statPassiveHomingState := NO_HOMING_ACTIVE;
    statExeOfHoming := CMD_BUSY;
    statBasicCommand := CMD_NO_SELECTION;
    statBasicCommandOld := CMD_NO_SELECTION;
    statBasicMotionState := NO_SELECTION;
    statExeOfBasicMotion := CMD_BUSY;
    statFirstCycleBasicMotion := FALSE;
    statApplicativeBasicMotionError := FALSE;
    statVelocityChangeOnTheFly := FALSE;
    statVelocity := 0.0;
    statAcceleration := 0.0;
    statAbortAcceleration := FALSE;
    statDeceleration := 0.0;
    statJerk := 0.0;

    statPositionControlled := TRUE;
    statFirstCycleDone := FALSE;

    statTorqueLimitingState := NO_TORQUE_LIMITING_ACTIVE;
    statTorqueLimitingErrorOld := FALSE;
    statTorqueLimit := -1.0;
    statJogMode := JOG_MODE_CONTINUOUS;
    statDirection := SPECIFIED_DIR;
    statHomingPosition         := 0.0;
    statHomingSubState         := HOMING_IDLE;
    statIncJogSubState         := INC_JOG_IDLE;
    statIncJogStartPosition    := 0.0;
    statIncJogDirectionOld     := 0;
    statIncrement              := 0.0;
    statIncJogDistance         := 0.0;
    statResetIncJog            := TRUE;
    statPosition               := 0.0;
    statPositionChangeOnTheFly := FALSE;

    statHomingMode                   := DIRECT_HOMING;
    statActiveHomingState            := NO_HOMING_ACTIVE;
    statSupImpCommand                := CMD_NO_SELECTION;
    statSupImpCommandOld             := CMD_NO_SELECTION;
    statSupImpMotionState            := NO_SELECTION;
    statExeOfSupImpMotionState       := CMD_BUSY;
    statFirstCycleSupImpMotion       := FALSE;
    statSupImpMotionPosition         := 0.0;
    statApplicativeSupImpMotionError := FALSE;
    statRatioChangeOnTheFly          := FALSE;
    statChangePhaseShiftOnTheFly     := FALSE;
    statPhaseShift                   := 0.0;
    statPhaseAbsolute                := TRUE;
    statRatioNumerator               := 0;
    statRatioDenominator             := 0;

   (* Tags for synchronized motion simulation*)
    statEnableAxis := FALSE;
    statSyncMotionSimulationState  := AXIS_NOT_IN_SIM;
    statSynchronizedMotionErrorOld := FALSE;
    statMainSelectionState := 0;
    statMasterSyncPosition := 0.0;
    statSlaveSyncPosition := 0.0;
    statSyncDirection := FORWARD_DIR;
    statMasterStartDistance := 0.0;
    statSyncProfileReference := 0;
    statApplicationMode := 0;

   (* ===========================================================*)
   (* Disable Axis*)
    IF (instPower.Busy = TRUE) THEN
        instPower(Axis := axis,
                  Enable := FALSE,
                  Enable_Positive := FALSE,
                  Enable_Negative := FALSE,
        (*StartMode :=  configuration.power.startMode,
	                   StopMode :=  configuration.power.stopMode*) );

       (* Check if error occurred*)
        IF (instPower.Error = TRUE) THEN
           (*Write only diagnostics IF error occurred AT falling edge OF MC_POWER*)
            diagnostics.status                  := ERR_MC_POWER;
            diagnostics.subfunctionStatus       := instPower.ErrorId;
            diagnostics.basicMotionState        := statBasicMotionState;
            diagnostics.superimposedMotionState := statSupImpMotionState;
        END_IF;
    END_IF;

   (* Set old value of enable for edge detection and end execution*)
    statEnableOld := enable;
    RETURN;
    {END_REGION}

   (* Check if FB is enabled - first cycle*)
ELSIF enable AND NOT statEnableOld THEN
    {REGION "FB_RISING_EDGE_AT_ENABLE_FB"}
   (* Busy is set at rising edge of enable input*)
    busy   := TRUE;
    status := STATUS_FB_FIRST_CALL;
   (* StatStatus will be written in next cycle*)
    statStatus := STATUS_SUBSEQUENT_CALL;

   (* Reset error and diagnostics outputs*)
    statErrorUserCleared := FALSE;
    statErrorAutoCleared := FALSE;
    diagnostics          := statEmptyDiagnostics;
    statDiagnostics      := statEmptyDiagnostics;

   (* Copy inputs*)
    statExtendedCommand.0 := resetAxis;
    statBasicCommand.8    := gearInAbsolute;
    statBasicCommand.9    := camIn;
    statSupImpCommand.1   := phasing;
    statBasicCommand.7    := gearInRelative;
    statBasicCommand.5    := posRelative;
    statBasicCommand.6    := posAbsolute;
    statSupImpCommand.0   := posSuperimposed;
    statSupImpCommandOld  := statSupImpCommand;
   (*  statExtendedCommand.1 :=  torqueLimiting;  // V1.0.2 Removed for activation at FB Enable *)

    statBasicCommand.0  := fastStop;
    statBasicCommand.1  := stop;
    statBasicCommand.2  := jogForward;
    statBasicCommand.3  := jogBackward;
    statBasicCommand.4  := moveVelocity;
    statBasicCommandOld := statBasicCommand;
   (* Set old value of homing input*)
    statHomingOld := homing;

    statExtendedCommandOld := statExtendedCommand;
   (* Set old value of enable for edge detection and end execution*)
    statEnableOld := enable;
    RETURN;
    {END_REGION}

   (* Check if function block is disabled or UserClearedError is present*)
ELSIF NOT enable OR statErrorUserCleared THEN
    {REGION "FB_DISABLED"}
    IF (enable = FALSE) THEN
        status := STATUS_NO_CALL;
    END_IF;

   (* Disable Axis*)
    IF (instPower.Busy = TRUE) THEN
        instPower(Axis := axis,
                  Enable := FALSE,
                  Enable_Positive := TRUE,
                  Enable_Negative := TRUE,
        (*StartMode :=  configuration.power.startMode,
	                   StopMode :=  configuration.power.stopMode*) );

       (* Check if error occurred*)
        IF (instPower.Error = TRUE) THEN
            diagnostics.status                  := ERR_MC_POWER;
            diagnostics.subfunctionStatus       := instPower.ErrorId;
            diagnostics.basicMotionState        := statBasicMotionState;
            diagnostics.superimposedMotionState := statSupImpMotionState;
        END_IF;
    ELSE
       (* V1.00.03 Reset if torque limiting is busy and axis is disabled *)
        IF (instTorqueLimiting.Busy = TRUE) THEN
            instTorqueLimiting(Axis := axis,
                               Enable := FALSE);
        ELSE
            busy := FALSE;
        END_IF;
    END_IF;

    statEnableOld := enable;
    RETURN;
    {END_REGION}

ELSE
    {REGION "FB_ENABLED"}
   (* Copy extended inputs*)
    statExtendedCommand.0 := resetAxis;
    tempEnableAxis        := enableAxis;
    statExtendedCommand.1 := torqueLimiting;
    statBasicCommand.0    := fastStop;
    statBasicCommand.1    := stop;
    statBasicCommand.2    := jogForward;
    statBasicCommand.3    := jogBackward;
    statBasicCommand.4    := moveVelocity;
    statBasicCommand.5    := posRelative;
    statBasicCommand.6    := posAbsolute;
    statSupImpCommand.0   := posSuperimposed;
    tempHoming            := homing;
    IF (tempHoming = TRUE) AND (statHomingOld = FALSE)
        THEN
       (* Rising edge on homing input*)
        statExtendedCommand.2 := TRUE;
        IF (configuration.homing.extendedMode = HOMING_ON_FIXED_STOP) OR(* Extended Homing mode (active)*)
            (configuration.homing.extendedMode = -1) AND
            ((configuration.homing.mode = ACTIVE_HOMING) OR (configuration.homing.mode = ACTIVE_HOMING_TO_DEF_VALUE))
            THEN
            ;                             (* Active Homing selected*)
            statBasicCommand.10   := TRUE;(* Cmd is BasicMotionCmd*)
            statExtendedCommand.2 := FALSE;
        ELSE
            ;(* Passive Homing selected*)
           (* Bit in extended cmd already written*)
        END_IF;

    ELSIF (tempHoming = FALSE) AND (statHomingOld = TRUE)
        THEN
       (* Falling edge on homing input*)
        statExtendedCommand.2 := FALSE;
        statBasicCommand.10   := FALSE;

    ELSE
        ;(* Do nothing - wait for rising / Falling edge*)
    END_IF;

    statBasicCommand.7  := gearInRelative;
    statBasicCommand.8  := gearInAbsolute;
    statBasicCommand.9  := camIn;
    statSupImpCommand.1 := phasing;

   (* Statemachine for synchronized motion simulation*)
    {REGION "SYNCHRONIZED_MOTION_SIMULATION"}
    REPEAT
        tempStateChangeActive := FALSE;
        CASE statSyncMotionSimulationState OF
            AXIS_NOT_IN_SIM:

                (* Axis NOT in simulation*)
                (* ----------------------------------------------------------*)
                (* Enable SynchronizedMotionSimulation*)
                (*  instSyncMotionSimulation(Slave :=  axis, // V01.00.03 Dont Call synchronizedmotionSimulation if not active*)
                (*                           Enable := FALSE);*)
                (* ----------------------------------------------------------*)

